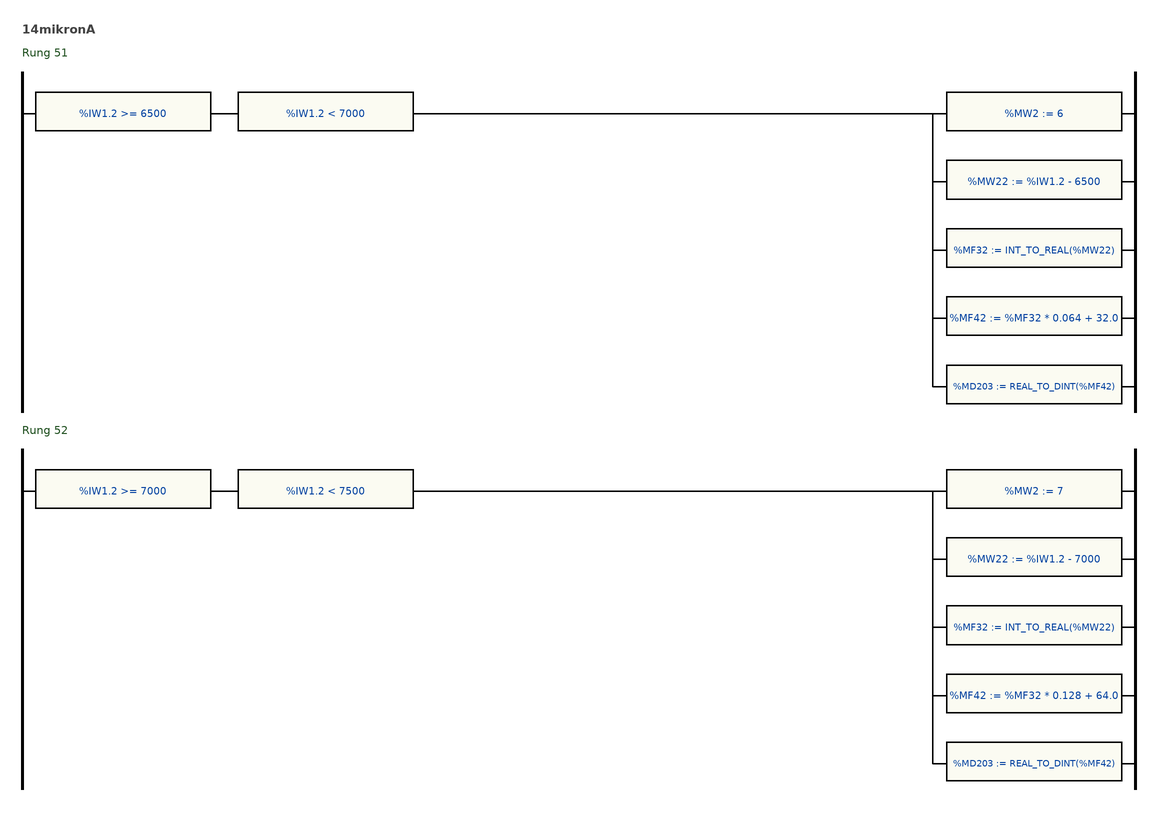
[picture p24: 14mikronA, ladder]

// Rung 51
  LD [ %IW1.2 >= 6500 ]
  AND [ %IW1.2 < 7000 ]
  [ %MW2 := 6 ]
  [ %MW22 := %IW1.2 - 6500 ]
  [ %MF32 := INT_TO_REAL ( %MW22 ) ]
  [ %MF42 := %MF32 * 0.064 + 32.0 ]
  [ %MD203 := REAL_TO_DINT ( %MF42 ) ]
  // as ST:
  //   IF %IW1.2 >= 6500 AND %IW1.2 < 7000 THEN %MW2 := 6; END_IF;
  //   IF %IW1.2 >= 6500 AND %IW1.2 < 7000 THEN %MW22 := %IW1.2 - 6500; END_IF;
  //   IF %IW1.2 >= 6500 AND %IW1.2 < 7000 THEN %MF32 := INT_TO_REAL ( %MW22 ); END_IF;
  //   IF %IW1.2 >= 6500 AND %IW1.2 < 7000 THEN %MF42 := %MF32 * 0.064 + 32.0; END_IF;
  //   IF %IW1.2 >= 6500 AND %IW1.2 < 7000 THEN %MD203 := REAL_TO_DINT ( %MF42 ); END_IF;

// Rung 52
  LD [ %IW1.2 >= 7000 ]
  AND [ %IW1.2 < 7500 ]
  [ %MW2 := 7 ]
  [ %MW22 := %IW1.2 - 7000 ]
  [ %MF32 := INT_TO_REAL ( %MW22 ) ]
  [ %MF42 := %MF32 * 0.128 + 64.0 ]
  [ %MD203 := REAL_TO_DINT ( %MF42 ) ]
  // as ST:
  //   IF %IW1.2 >= 7000 AND %IW1.2 < 7500 THEN %MW2 := 7; END_IF;
  //   IF %IW1.2 >= 7000 AND %IW1.2 < 7500 THEN %MW22 := %IW1.2 - 7000; END_IF;
  //   IF %IW1.2 >= 7000 AND %IW1.2 < 7500 THEN %MF32 := INT_TO_REAL ( %MW22 ); END_IF;
  //   IF %IW1.2 >= 7000 AND %IW1.2 < 7500 THEN %MF42 := %MF32 * 0.128 + 64.0; END_IF;
  //   IF %IW1.2 >= 7000 AND %IW1.2 < 7500 THEN %MD203 := REAL_TO_DINT ( %MF42 ); END_IF;

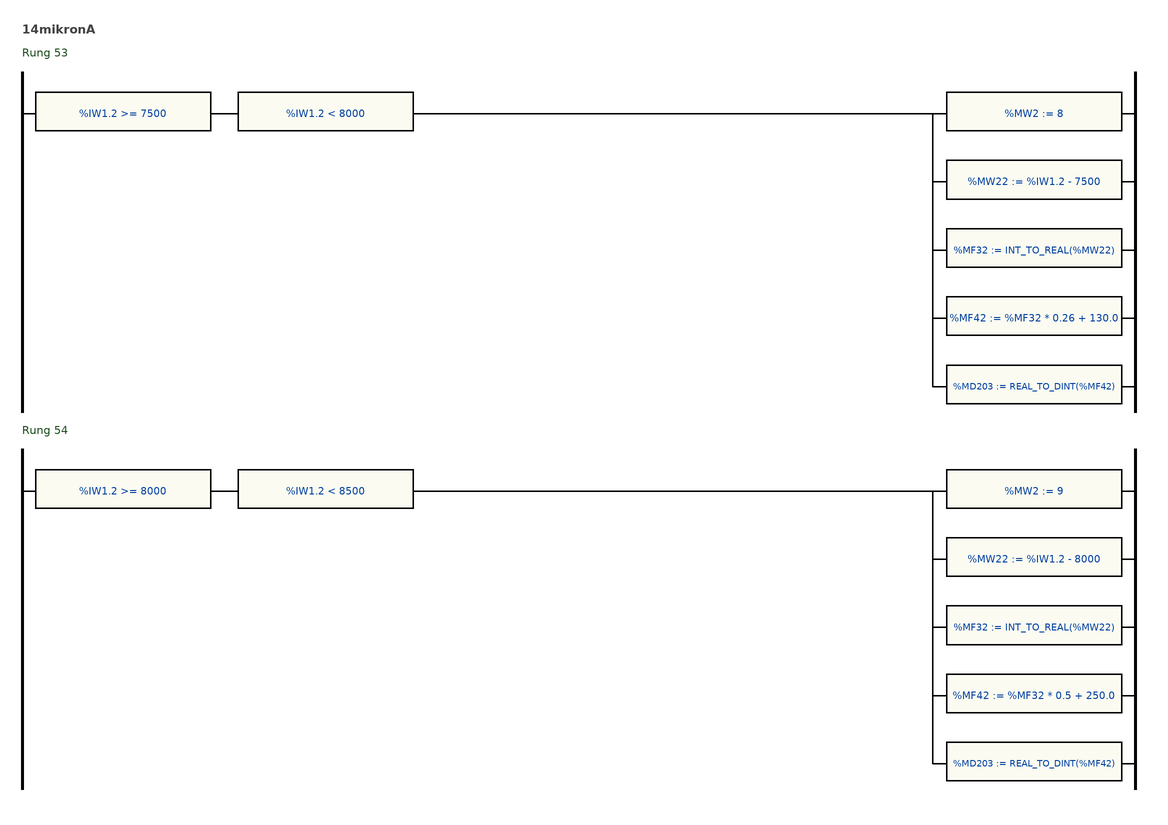

// Rung 53
  LD [ %IW1.2 >= 7500 ]
  AND [ %IW1.2 < 8000 ]
  [ %MW2 := 8 ]
  [ %MW22 := %IW1.2 - 7500 ]
  [ %MF32 := INT_TO_REAL ( %MW22 ) ]
  [ %MF42 := %MF32 * 0.26 + 130.0 ]
  [ %MD203 := REAL_TO_DINT ( %MF42 ) ]
  // as ST:
  //   IF %IW1.2 >= 7500 AND %IW1.2 < 8000 THEN %MW2 := 8; END_IF;
  //   IF %IW1.2 >= 7500 AND %IW1.2 < 8000 THEN %MW22 := %IW1.2 - 7500; END_IF;
  //   IF %IW1.2 >= 7500 AND %IW1.2 < 8000 THEN %MF32 := INT_TO_REAL ( %MW22 ); END_IF;
  //   IF %IW1.2 >= 7500 AND %IW1.2 < 8000 THEN %MF42 := %MF32 * 0.26 + 130.0; END_IF;
  //   IF %IW1.2 >= 7500 AND %IW1.2 < 8000 THEN %MD203 := REAL_TO_DINT ( %MF42 ); END_IF;

// Rung 54
  LD [ %IW1.2 >= 8000 ]
  AND [ %IW1.2 < 8500 ]
  [ %MW2 := 9 ]
  [ %MW22 := %IW1.2 - 8000 ]
  [ %MF32 := INT_TO_REAL ( %MW22 ) ]
  [ %MF42 := %MF32 * 0.5 + 250.0 ]
  [ %MD203 := REAL_TO_DINT ( %MF42 ) ]
  // as ST:
  //   IF %IW1.2 >= 8000 AND %IW1.2 < 8500 THEN %MW2 := 9; END_IF;
  //   IF %IW1.2 >= 8000 AND %IW1.2 < 8500 THEN %MW22 := %IW1.2 - 8000; END_IF;
  //   IF %IW1.2 >= 8000 AND %IW1.2 < 8500 THEN %MF32 := INT_TO_REAL ( %MW22 ); END_IF;
  //   IF %IW1.2 >= 8000 AND %IW1.2 < 8500 THEN %MF42 := %MF32 * 0.5 + 250.0; END_IF;
  //   IF %IW1.2 >= 8000 AND %IW1.2 < 8500 THEN %MD203 := REAL_TO_DINT ( %MF42 ); END_IF;

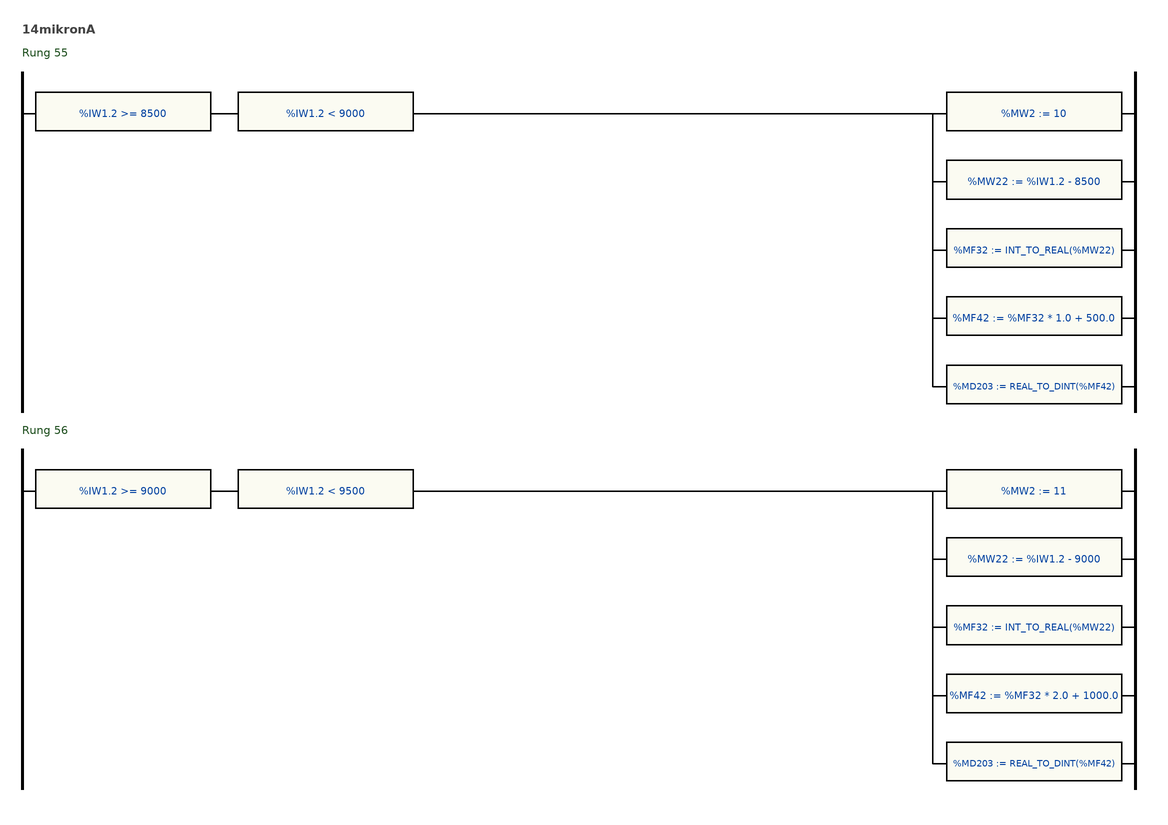

// Rung 55
  LD [ %IW1.2 >= 8500 ]
  AND [ %IW1.2 < 9000 ]
  [ %MW2 := 10 ]
  [ %MW22 := %IW1.2 - 8500 ]
  [ %MF32 := INT_TO_REAL ( %MW22 ) ]
  [ %MF42 := %MF32 * 1.0 + 500.0 ]
  [ %MD203 := REAL_TO_DINT ( %MF42 ) ]
  // as ST:
  //   IF %IW1.2 >= 8500 AND %IW1.2 < 9000 THEN %MW2 := 10; END_IF;
  //   IF %IW1.2 >= 8500 AND %IW1.2 < 9000 THEN %MW22 := %IW1.2 - 8500; END_IF;
  //   IF %IW1.2 >= 8500 AND %IW1.2 < 9000 THEN %MF32 := INT_TO_REAL ( %MW22 ); END_IF;
  //   IF %IW1.2 >= 8500 AND %IW1.2 < 9000 THEN %MF42 := %MF32 * 1.0 + 500.0; END_IF;
  //   IF %IW1.2 >= 8500 AND %IW1.2 < 9000 THEN %MD203 := REAL_TO_DINT ( %MF42 ); END_IF;

// Rung 56
  LD [ %IW1.2 >= 9000 ]
  AND [ %IW1.2 < 9500 ]
  [ %MW2 := 11 ]
  [ %MW22 := %IW1.2 - 9000 ]
  [ %MF32 := INT_TO_REAL ( %MW22 ) ]
  [ %MF42 := %MF32 * 2.0 + 1000.0 ]
  [ %MD203 := REAL_TO_DINT ( %MF42 ) ]
  // as ST:
  //   IF %IW1.2 >= 9000 AND %IW1.2 < 9500 THEN %MW2 := 11; END_IF;
  //   IF %IW1.2 >= 9000 AND %IW1.2 < 9500 THEN %MW22 := %IW1.2 - 9000; END_IF;
  //   IF %IW1.2 >= 9000 AND %IW1.2 < 9500 THEN %MF32 := INT_TO_REAL ( %MW22 ); END_IF;
  //   IF %IW1.2 >= 9000 AND %IW1.2 < 9500 THEN %MF42 := %MF32 * 2.0 + 1000.0; END_IF;
  //   IF %IW1.2 >= 9000 AND %IW1.2 < 9500 THEN %MD203 := REAL_TO_DINT ( %MF42 ); END_IF;

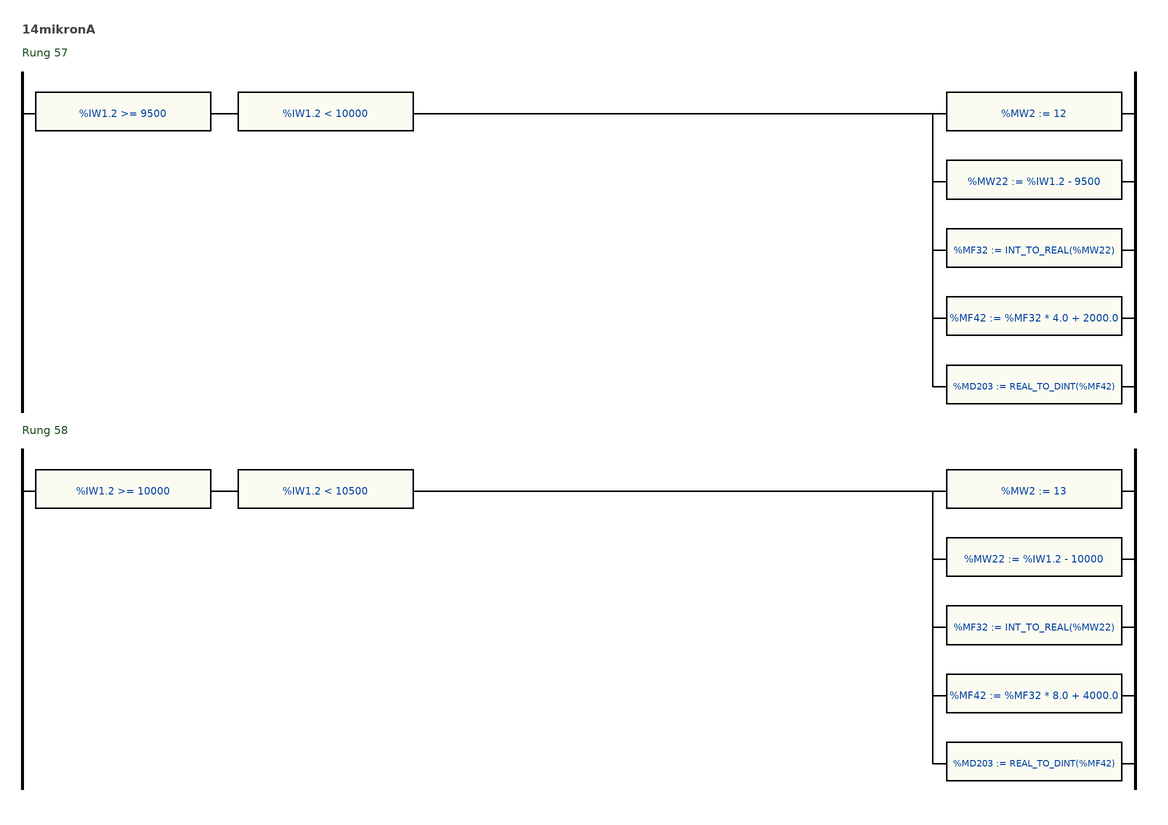

// Rung 57
  LD [ %IW1.2 >= 9500 ]
  AND [ %IW1.2 < 10000 ]
  [ %MW2 := 12 ]
  [ %MW22 := %IW1.2 - 9500 ]
  [ %MF32 := INT_TO_REAL ( %MW22 ) ]
  [ %MF42 := %MF32 * 4.0 + 2000.0 ]
  [ %MD203 := REAL_TO_DINT ( %MF42 ) ]
  // as ST:
  //   IF %IW1.2 >= 9500 AND %IW1.2 < 10000 THEN %MW2 := 12; END_IF;
  //   IF %IW1.2 >= 9500 AND %IW1.2 < 10000 THEN %MW22 := %IW1.2 - 9500; END_IF;
  //   IF %IW1.2 >= 9500 AND %IW1.2 < 10000 THEN %MF32 := INT_TO_REAL ( %MW22 ); END_IF;
  //   IF %IW1.2 >= 9500 AND %IW1.2 < 10000 THEN %MF42 := %MF32 * 4.0 + 2000.0; END_IF;
  //   IF %IW1.2 >= 9500 AND %IW1.2 < 10000 THEN %MD203 := REAL_TO_DINT ( %MF42 ); END_IF;

// Rung 58
  LD [ %IW1.2 >= 10000 ]
  AND [ %IW1.2 < 10500 ]
  [ %MW2 := 13 ]
  [ %MW22 := %IW1.2 - 10000 ]
  [ %MF32 := INT_TO_REAL ( %MW22 ) ]
  [ %MF42 := %MF32 * 8.0 + 4000.0 ]
  [ %MD203 := REAL_TO_DINT ( %MF42 ) ]
  // as ST:
  //   IF %IW1.2 >= 10000 AND %IW1.2 < 10500 THEN %MW2 := 13; END_IF;
  //   IF %IW1.2 >= 10000 AND %IW1.2 < 10500 THEN %MW22 := %IW1.2 - 10000; END_IF;
  //   IF %IW1.2 >= 10000 AND %IW1.2 < 10500 THEN %MF32 := INT_TO_REAL ( %MW22 ); END_IF;
  //   IF %IW1.2 >= 10000 AND %IW1.2 < 10500 THEN %MF42 := %MF32 * 8.0 + 4000.0; END_IF;
  //   IF %IW1.2 >= 10000 AND %IW1.2 < 10500 THEN %MD203 := REAL_TO_DINT ( %MF42 ); END_IF;

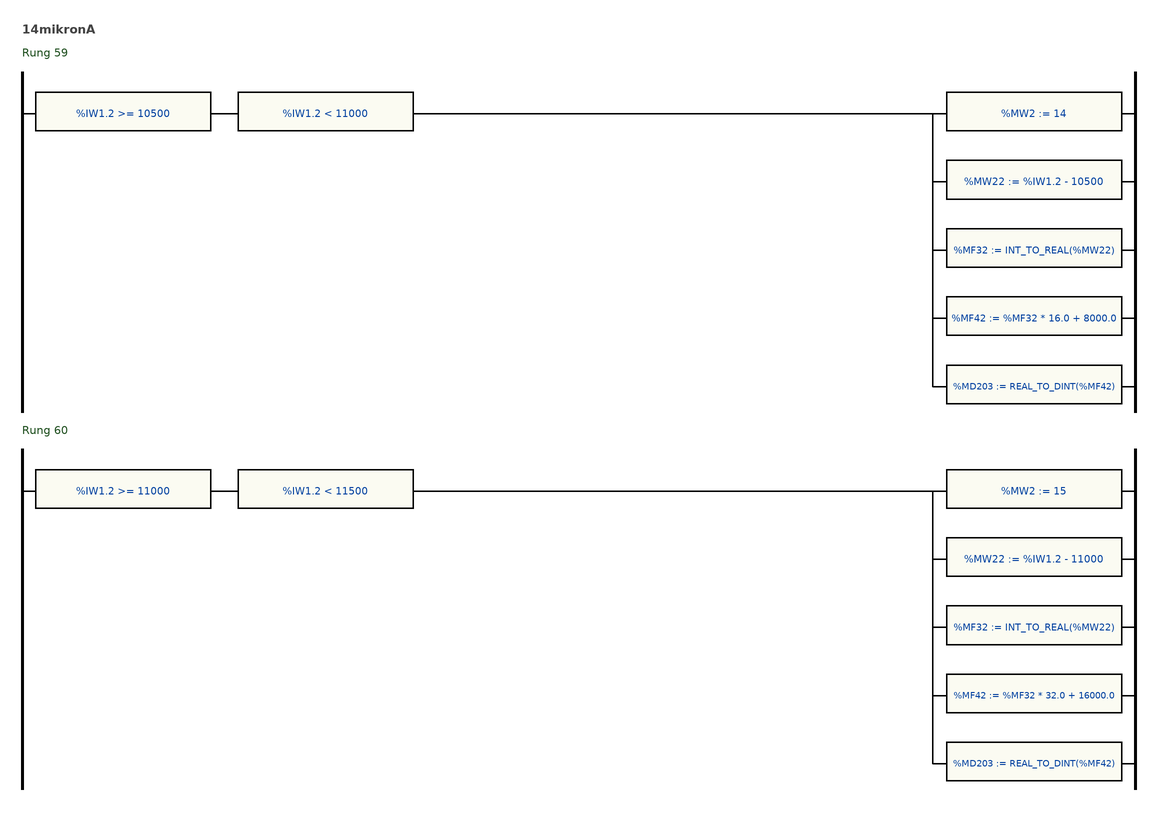

// Rung 59
  LD [ %IW1.2 >= 10500 ]
  AND [ %IW1.2 < 11000 ]
  [ %MW2 := 14 ]
  [ %MW22 := %IW1.2 - 10500 ]
  [ %MF32 := INT_TO_REAL ( %MW22 ) ]
  [ %MF42 := %MF32 * 16.0 + 8000.0 ]
  [ %MD203 := REAL_TO_DINT ( %MF42 ) ]
  // as ST:
  //   IF %IW1.2 >= 10500 AND %IW1.2 < 11000 THEN %MW2 := 14; END_IF;
  //   IF %IW1.2 >= 10500 AND %IW1.2 < 11000 THEN %MW22 := %IW1.2 - 10500; END_IF;
  //   IF %IW1.2 >= 10500 AND %IW1.2 < 11000 THEN %MF32 := INT_TO_REAL ( %MW22 ); END_IF;
  //   IF %IW1.2 >= 10500 AND %IW1.2 < 11000 THEN %MF42 := %MF32 * 16.0 + 8000.0; END_IF;
  //   IF %IW1.2 >= 10500 AND %IW1.2 < 11000 THEN %MD203 := REAL_TO_DINT ( %MF42 ); END_IF;

// Rung 60
  LD [ %IW1.2 >= 11000 ]
  AND [ %IW1.2 < 11500 ]
  [ %MW2 := 15 ]
  [ %MW22 := %IW1.2 - 11000 ]
  [ %MF32 := INT_TO_REAL ( %MW22 ) ]
  [ %MF42 := %MF32 * 32.0 + 16000.0 ]
  [ %MD203 := REAL_TO_DINT ( %MF42 ) ]
  // as ST:
  //   IF %IW1.2 >= 11000 AND %IW1.2 < 11500 THEN %MW2 := 15; END_IF;
  //   IF %IW1.2 >= 11000 AND %IW1.2 < 11500 THEN %MW22 := %IW1.2 - 11000; END_IF;
  //   IF %IW1.2 >= 11000 AND %IW1.2 < 11500 THEN %MF32 := INT_TO_REAL ( %MW22 ); END_IF;
  //   IF %IW1.2 >= 11000 AND %IW1.2 < 11500 THEN %MF42 := %MF32 * 32.0 + 16000.0; END_IF;
  //   IF %IW1.2 >= 11000 AND %IW1.2 < 11500 THEN %MD203 := REAL_TO_DINT ( %MF42 ); END_IF;

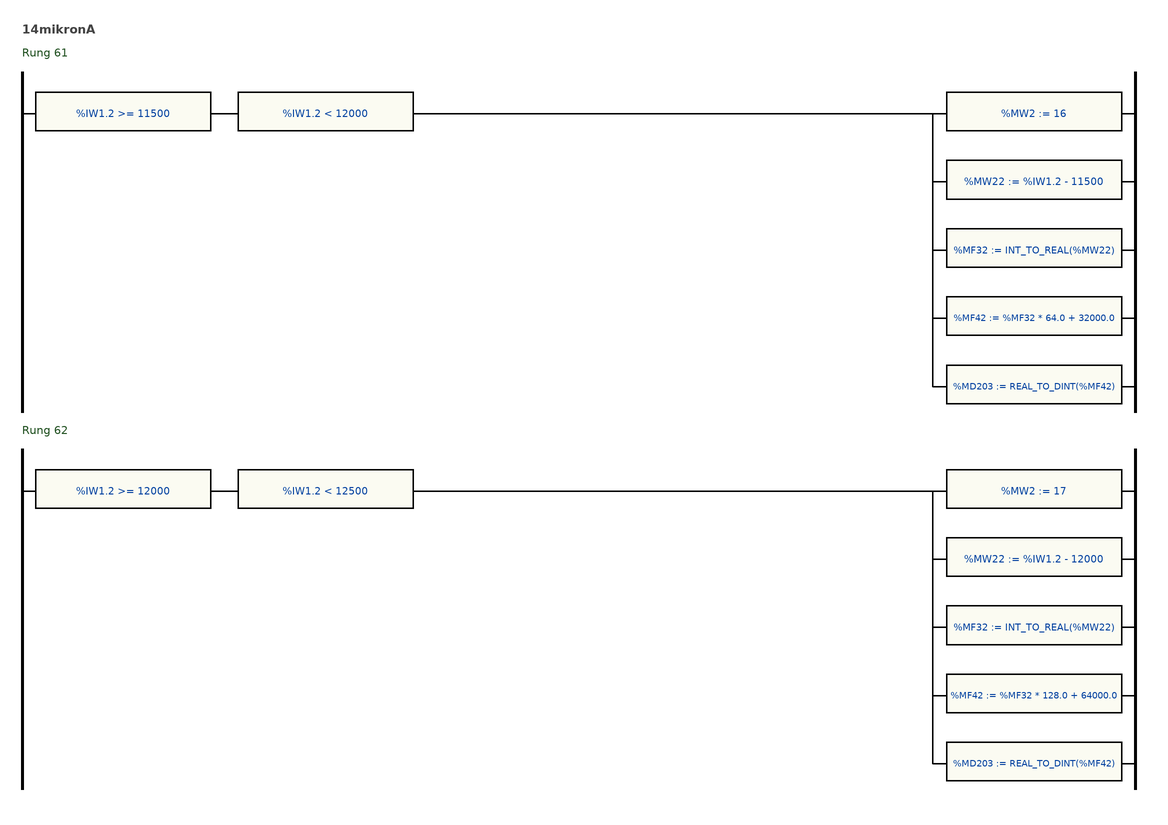

// Rung 61
  LD [ %IW1.2 >= 11500 ]
  AND [ %IW1.2 < 12000 ]
  [ %MW2 := 16 ]
  [ %MW22 := %IW1.2 - 11500 ]
  [ %MF32 := INT_TO_REAL ( %MW22 ) ]
  [ %MF42 := %MF32 * 64.0 + 32000.0 ]
  [ %MD203 := REAL_TO_DINT ( %MF42 ) ]
  // as ST:
  //   IF %IW1.2 >= 11500 AND %IW1.2 < 12000 THEN %MW2 := 16; END_IF;
  //   IF %IW1.2 >= 11500 AND %IW1.2 < 12000 THEN %MW22 := %IW1.2 - 11500; END_IF;
  //   IF %IW1.2 >= 11500 AND %IW1.2 < 12000 THEN %MF32 := INT_TO_REAL ( %MW22 ); END_IF;
  //   IF %IW1.2 >= 11500 AND %IW1.2 < 12000 THEN %MF42 := %MF32 * 64.0 + 32000.0; END_IF;
  //   IF %IW1.2 >= 11500 AND %IW1.2 < 12000 THEN %MD203 := REAL_TO_DINT ( %MF42 ); END_IF;

// Rung 62
  LD [ %IW1.2 >= 12000 ]
  AND [ %IW1.2 < 12500 ]
  [ %MW2 := 17 ]
  [ %MW22 := %IW1.2 - 12000 ]
  [ %MF32 := INT_TO_REAL ( %MW22 ) ]
  [ %MF42 := %MF32 * 128.0 + 64000.0 ]
  [ %MD203 := REAL_TO_DINT ( %MF42 ) ]
  // as ST:
  //   IF %IW1.2 >= 12000 AND %IW1.2 < 12500 THEN %MW2 := 17; END_IF;
  //   IF %IW1.2 >= 12000 AND %IW1.2 < 12500 THEN %MW22 := %IW1.2 - 12000; END_IF;
  //   IF %IW1.2 >= 12000 AND %IW1.2 < 12500 THEN %MF32 := INT_TO_REAL ( %MW22 ); END_IF;
  //   IF %IW1.2 >= 12000 AND %IW1.2 < 12500 THEN %MF42 := %MF32 * 128.0 + 64000.0; END_IF;
  //   IF %IW1.2 >= 12000 AND %IW1.2 < 12500 THEN %MD203 := REAL_TO_DINT ( %MF42 ); END_IF;

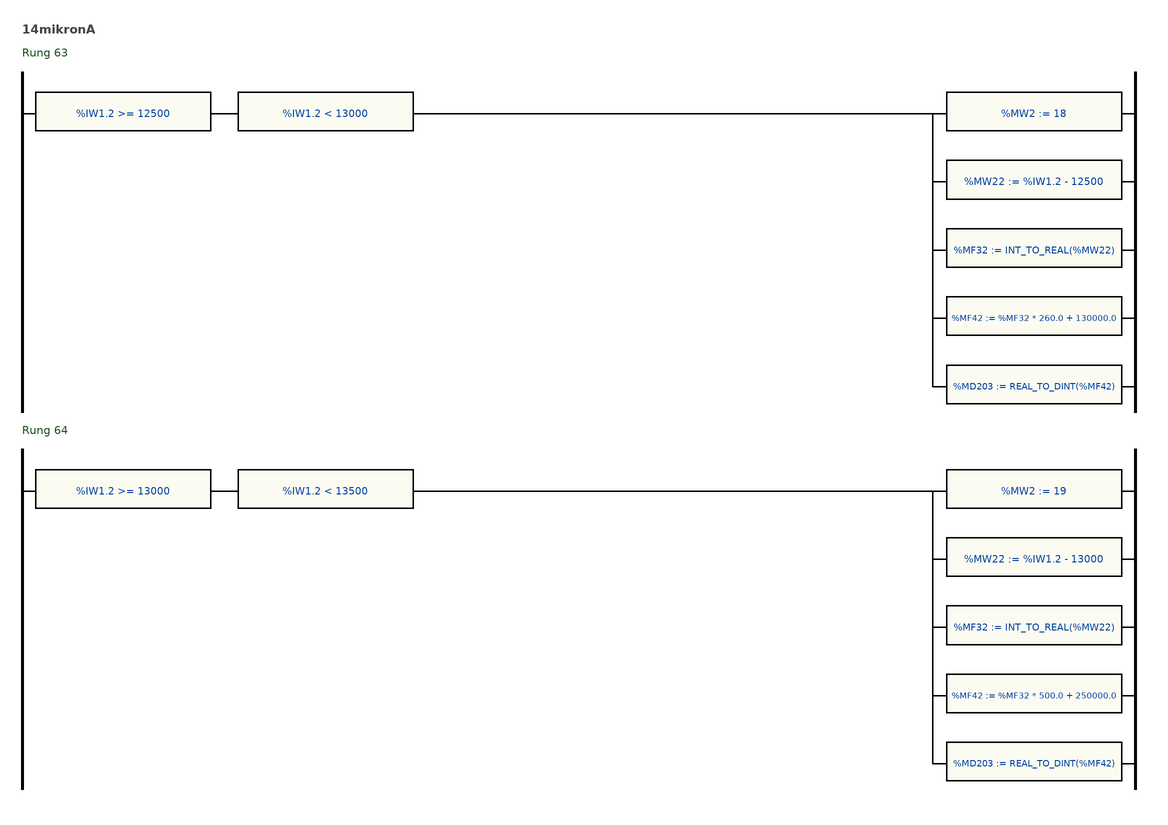

// Rung 63
  LD [ %IW1.2 >= 12500 ]
  AND [ %IW1.2 < 13000 ]
  [ %MW2 := 18 ]
  [ %MW22 := %IW1.2 - 12500 ]
  [ %MF32 := INT_TO_REAL ( %MW22 ) ]
  [ %MF42 := %MF32 * 260.0 + 130000.0 ]
  [ %MD203 := REAL_TO_DINT ( %MF42 ) ]
  // as ST:
  //   IF %IW1.2 >= 12500 AND %IW1.2 < 13000 THEN %MW2 := 18; END_IF;
  //   IF %IW1.2 >= 12500 AND %IW1.2 < 13000 THEN %MW22 := %IW1.2 - 12500; END_IF;
  //   IF %IW1.2 >= 12500 AND %IW1.2 < 13000 THEN %MF32 := INT_TO_REAL ( %MW22 ); END_IF;
  //   IF %IW1.2 >= 12500 AND %IW1.2 < 13000 THEN %MF42 := %MF32 * 260.0 + 130000.0; END_IF;
  //   IF %IW1.2 >= 12500 AND %IW1.2 < 13000 THEN %MD203 := REAL_TO_DINT ( %MF42 ); END_IF;

// Rung 64
  LD [ %IW1.2 >= 13000 ]
  AND [ %IW1.2 < 13500 ]
  [ %MW2 := 19 ]
  [ %MW22 := %IW1.2 - 13000 ]
  [ %MF32 := INT_TO_REAL ( %MW22 ) ]
  [ %MF42 := %MF32 * 500.0 + 250000.0 ]
  [ %MD203 := REAL_TO_DINT ( %MF42 ) ]
  // as ST:
  //   IF %IW1.2 >= 13000 AND %IW1.2 < 13500 THEN %MW2 := 19; END_IF;
  //   IF %IW1.2 >= 13000 AND %IW1.2 < 13500 THEN %MW22 := %IW1.2 - 13000; END_IF;
  //   IF %IW1.2 >= 13000 AND %IW1.2 < 13500 THEN %MF32 := INT_TO_REAL ( %MW22 ); END_IF;
  //   IF %IW1.2 >= 13000 AND %IW1.2 < 13500 THEN %MF42 := %MF32 * 500.0 + 250000.0; END_IF;
  //   IF %IW1.2 >= 13000 AND %IW1.2 < 13500 THEN %MD203 := REAL_TO_DINT ( %MF42 ); END_IF;

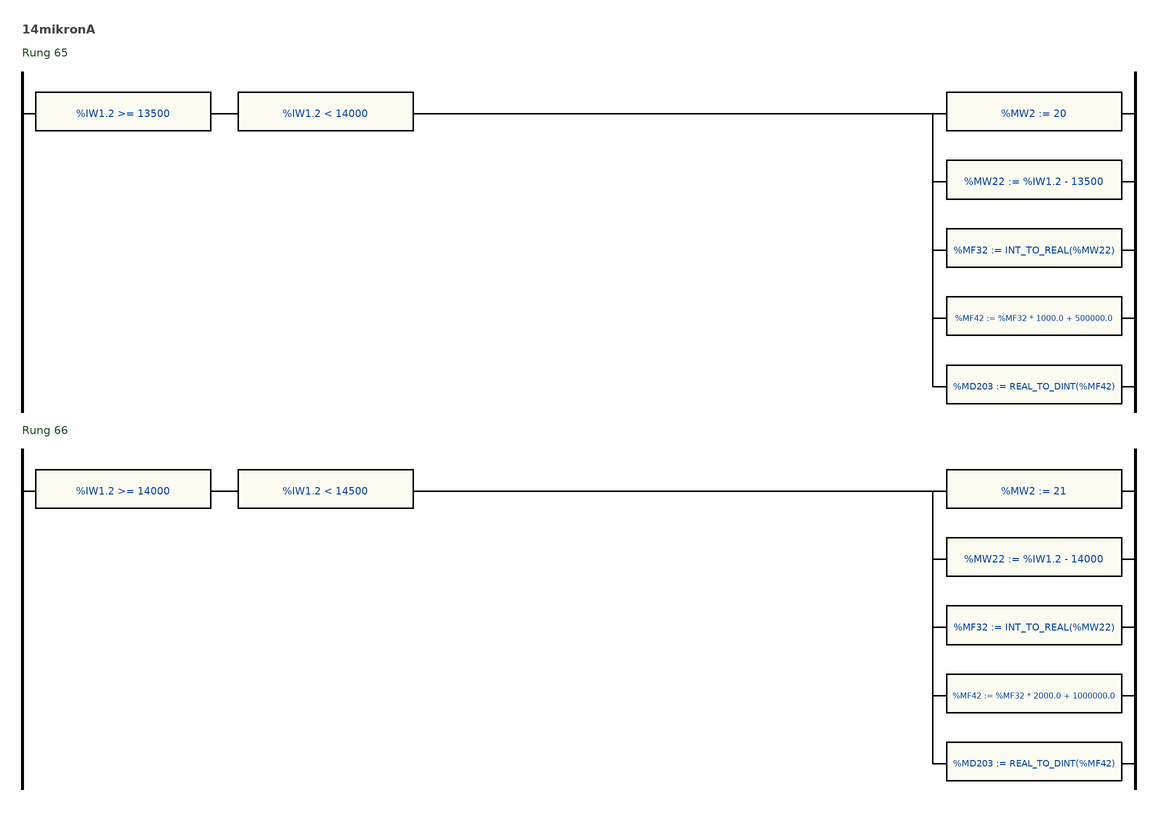

// Rung 65
  LD [ %IW1.2 >= 13500 ]
  AND [ %IW1.2 < 14000 ]
  [ %MW2 := 20 ]
  [ %MW22 := %IW1.2 - 13500 ]
  [ %MF32 := INT_TO_REAL ( %MW22 ) ]
  [ %MF42 := %MF32 * 1000.0 + 500000.0 ]
  [ %MD203 := REAL_TO_DINT ( %MF42 ) ]
  // as ST:
  //   IF %IW1.2 >= 13500 AND %IW1.2 < 14000 THEN %MW2 := 20; END_IF;
  //   IF %IW1.2 >= 13500 AND %IW1.2 < 14000 THEN %MW22 := %IW1.2 - 13500; END_IF;
  //   IF %IW1.2 >= 13500 AND %IW1.2 < 14000 THEN %MF32 := INT_TO_REAL ( %MW22 ); END_IF;
  //   IF %IW1.2 >= 13500 AND %IW1.2 < 14000 THEN %MF42 := %MF32 * 1000.0 + 500000.0; END_IF;
  //   IF %IW1.2 >= 13500 AND %IW1.2 < 14000 THEN %MD203 := REAL_TO_DINT ( %MF42 ); END_IF;

// Rung 66
  LD [ %IW1.2 >= 14000 ]
  AND [ %IW1.2 < 14500 ]
  [ %MW2 := 21 ]
  [ %MW22 := %IW1.2 - 14000 ]
  [ %MF32 := INT_TO_REAL ( %MW22 ) ]
  [ %MF42 := %MF32 * 2000.0 + 1000000.0 ]
  [ %MD203 := REAL_TO_DINT ( %MF42 ) ]
  // as ST:
  //   IF %IW1.2 >= 14000 AND %IW1.2 < 14500 THEN %MW2 := 21; END_IF;
  //   IF %IW1.2 >= 14000 AND %IW1.2 < 14500 THEN %MW22 := %IW1.2 - 14000; END_IF;
  //   IF %IW1.2 >= 14000 AND %IW1.2 < 14500 THEN %MF32 := INT_TO_REAL ( %MW22 ); END_IF;
  //   IF %IW1.2 >= 14000 AND %IW1.2 < 14500 THEN %MF42 := %MF32 * 2000.0 + 1000000.0; END_IF;
  //   IF %IW1.2 >= 14000 AND %IW1.2 < 14500 THEN %MD203 := REAL_TO_DINT ( %MF42 ); END_IF;

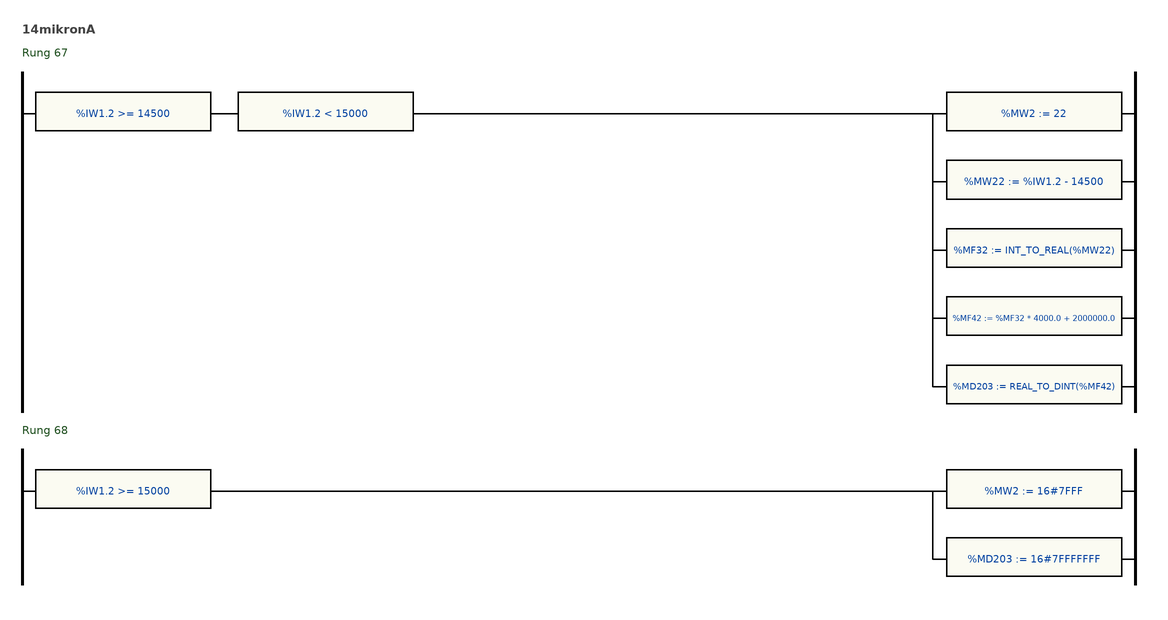

// Rung 67
  LD [ %IW1.2 >= 14500 ]
  AND [ %IW1.2 < 15000 ]
  [ %MW2 := 22 ]
  [ %MW22 := %IW1.2 - 14500 ]
  [ %MF32 := INT_TO_REAL ( %MW22 ) ]
  [ %MF42 := %MF32 * 4000.0 + 2000000.0 ]
  [ %MD203 := REAL_TO_DINT ( %MF42 ) ]
  // as ST:
  //   IF %IW1.2 >= 14500 AND %IW1.2 < 15000 THEN %MW2 := 22; END_IF;
  //   IF %IW1.2 >= 14500 AND %IW1.2 < 15000 THEN %MW22 := %IW1.2 - 14500; END_IF;
  //   IF %IW1.2 >= 14500 AND %IW1.2 < 15000 THEN %MF32 := INT_TO_REAL ( %MW22 ); END_IF;
  //   IF %IW1.2 >= 14500 AND %IW1.2 < 15000 THEN %MF42 := %MF32 * 4000.0 + 2000000.0; END_IF;
  //   IF %IW1.2 >= 14500 AND %IW1.2 < 15000 THEN %MD203 := REAL_TO_DINT ( %MF42 ); END_IF;

// Rung 68
  LD [ %IW1.2 >= 15000 ]
  [ %MW2 := 16#7FFF ]
  [ %MD203 := 16#7FFFFFFF ]
  // as ST:
  //   IF %IW1.2 >= 15000 THEN %MW2 := 16#7FFF; END_IF;
  //   IF %IW1.2 >= 15000 THEN %MD203 := 16#7FFFFFFF; END_IF;

POU 4mikronB
  (* SectionNumber=4 *)

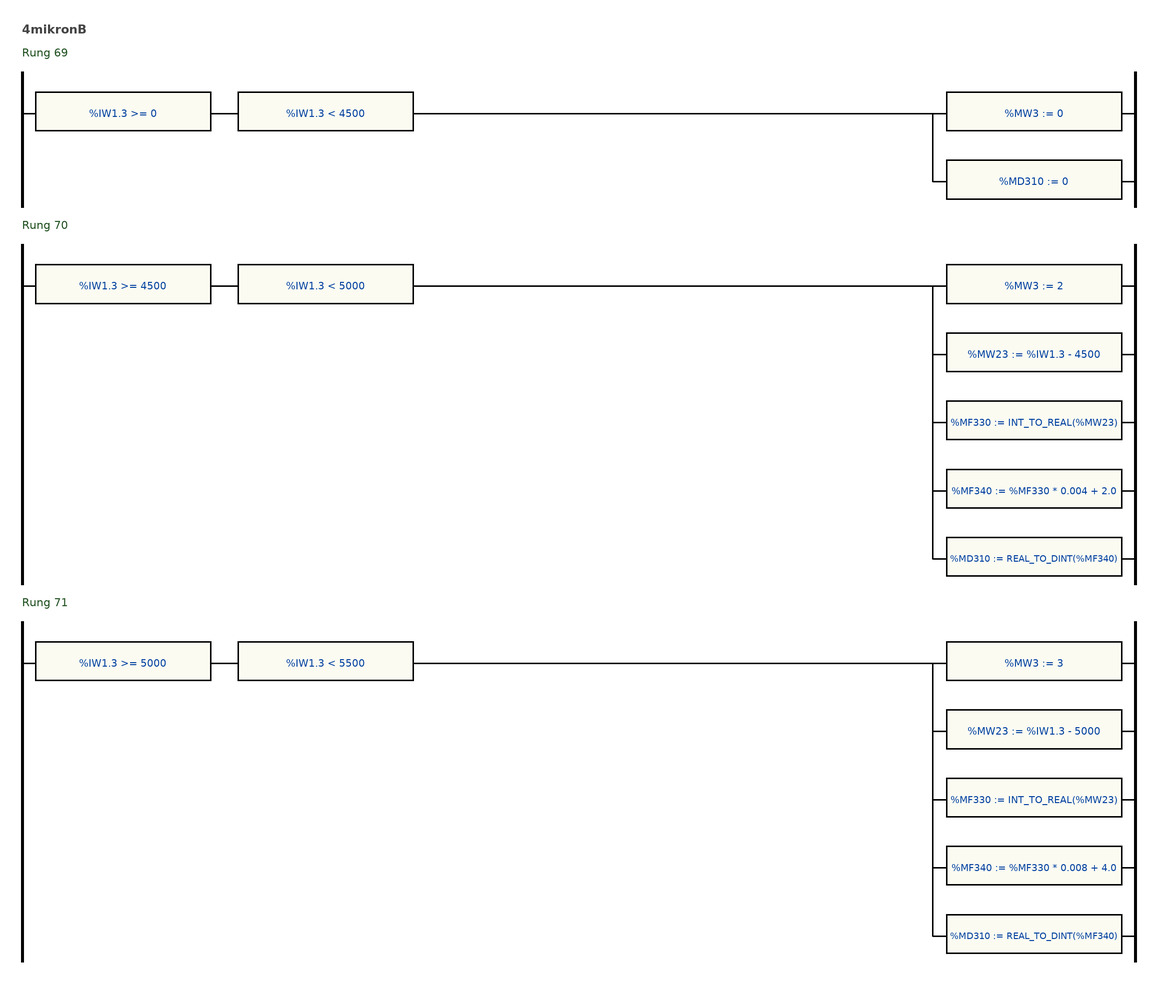

// Rung 69
  LD [ %IW1.3 >= 0 ]
  AND [ %IW1.3 < 4500 ]
  [ %MW3 := 0 ]
  [ %MD310 := 0 ]
  // as ST:
  //   IF %IW1.3 >= 0 AND %IW1.3 < 4500 THEN %MW3 := 0; END_IF;
  //   IF %IW1.3 >= 0 AND %IW1.3 < 4500 THEN %MD310 := 0; END_IF;

// Rung 70
  LD [ %IW1.3 >= 4500 ]
  AND [ %IW1.3 < 5000 ]
  [ %MW3 := 2 ]
  [ %MW23 := %IW1.3 - 4500 ]
  [ %MF330 := INT_TO_REAL ( %MW23 ) ]
  [ %MF340 := %MF330 * 0.004 + 2.0 ]
  [ %MD310 := REAL_TO_DINT ( %MF340 ) ]
  // as ST:
  //   IF %IW1.3 >= 4500 AND %IW1.3 < 5000 THEN %MW3 := 2; END_IF;
  //   IF %IW1.3 >= 4500 AND %IW1.3 < 5000 THEN %MW23 := %IW1.3 - 4500; END_IF;
  //   IF %IW1.3 >= 4500 AND %IW1.3 < 5000 THEN %MF330 := INT_TO_REAL ( %MW23 ); END_IF;
  //   IF %IW1.3 >= 4500 AND %IW1.3 < 5000 THEN %MF340 := %MF330 * 0.004 + 2.0; END_IF;
  //   IF %IW1.3 >= 4500 AND %IW1.3 < 5000 THEN %MD310 := REAL_TO_DINT ( %MF340 ); END_IF;

// Rung 71
  LD [ %IW1.3 >= 5000 ]
  AND [ %IW1.3 < 5500 ]
  [ %MW3 := 3 ]
  [ %MW23 := %IW1.3 - 5000 ]
  [ %MF330 := INT_TO_REAL ( %MW23 ) ]
  [ %MF340 := %MF330 * 0.008 + 4.0 ]
  [ %MD310 := REAL_TO_DINT ( %MF340 ) ]
  // as ST:
  //   IF %IW1.3 >= 5000 AND %IW1.3 < 5500 THEN %MW3 := 3; END_IF;
  //   IF %IW1.3 >= 5000 AND %IW1.3 < 5500 THEN %MW23 := %IW1.3 - 5000; END_IF;
  //   IF %IW1.3 >= 5000 AND %IW1.3 < 5500 THEN %MF330 := INT_TO_REAL ( %MW23 ); END_IF;
  //   IF %IW1.3 >= 5000 AND %IW1.3 < 5500 THEN %MF340 := %MF330 * 0.008 + 4.0; END_IF;
  //   IF %IW1.3 >= 5000 AND %IW1.3 < 5500 THEN %MD310 := REAL_TO_DINT ( %MF340 ); END_IF;

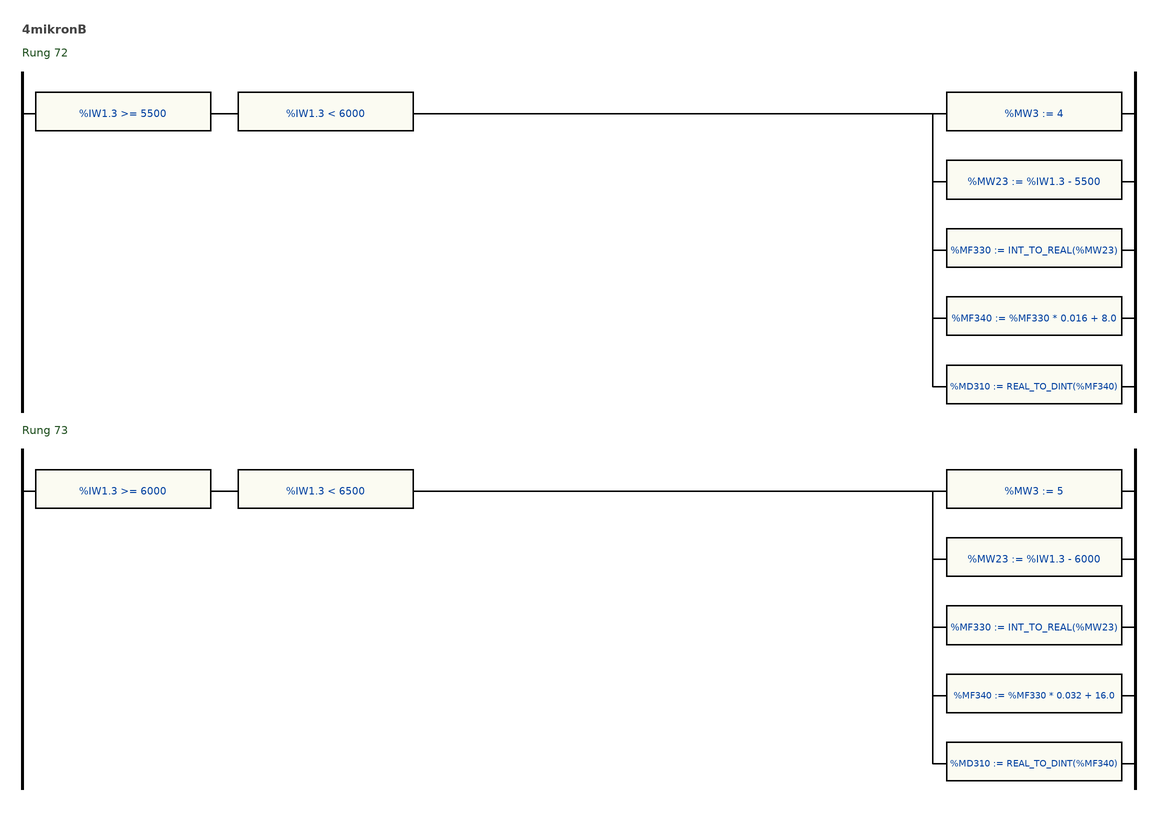

// Rung 72
  LD [ %IW1.3 >= 5500 ]
  AND [ %IW1.3 < 6000 ]
  [ %MW3 := 4 ]
  [ %MW23 := %IW1.3 - 5500 ]
  [ %MF330 := INT_TO_REAL ( %MW23 ) ]
  [ %MF340 := %MF330 * 0.016 + 8.0 ]
  [ %MD310 := REAL_TO_DINT ( %MF340 ) ]
  // as ST:
  //   IF %IW1.3 >= 5500 AND %IW1.3 < 6000 THEN %MW3 := 4; END_IF;
  //   IF %IW1.3 >= 5500 AND %IW1.3 < 6000 THEN %MW23 := %IW1.3 - 5500; END_IF;
  //   IF %IW1.3 >= 5500 AND %IW1.3 < 6000 THEN %MF330 := INT_TO_REAL ( %MW23 ); END_IF;
  //   IF %IW1.3 >= 5500 AND %IW1.3 < 6000 THEN %MF340 := %MF330 * 0.016 + 8.0; END_IF;
  //   IF %IW1.3 >= 5500 AND %IW1.3 < 6000 THEN %MD310 := REAL_TO_DINT ( %MF340 ); END_IF;

// Rung 73
  LD [ %IW1.3 >= 6000 ]
  AND [ %IW1.3 < 6500 ]
  [ %MW3 := 5 ]
  [ %MW23 := %IW1.3 - 6000 ]
  [ %MF330 := INT_TO_REAL ( %MW23 ) ]
  [ %MF340 := %MF330 * 0.032 + 16.0 ]
  [ %MD310 := REAL_TO_DINT ( %MF340 ) ]
  // as ST:
  //   IF %IW1.3 >= 6000 AND %IW1.3 < 6500 THEN %MW3 := 5; END_IF;
  //   IF %IW1.3 >= 6000 AND %IW1.3 < 6500 THEN %MW23 := %IW1.3 - 6000; END_IF;
  //   IF %IW1.3 >= 6000 AND %IW1.3 < 6500 THEN %MF330 := INT_TO_REAL ( %MW23 ); END_IF;
  //   IF %IW1.3 >= 6000 AND %IW1.3 < 6500 THEN %MF340 := %MF330 * 0.032 + 16.0; END_IF;
  //   IF %IW1.3 >= 6000 AND %IW1.3 < 6500 THEN %MD310 := REAL_TO_DINT ( %MF340 ); END_IF;

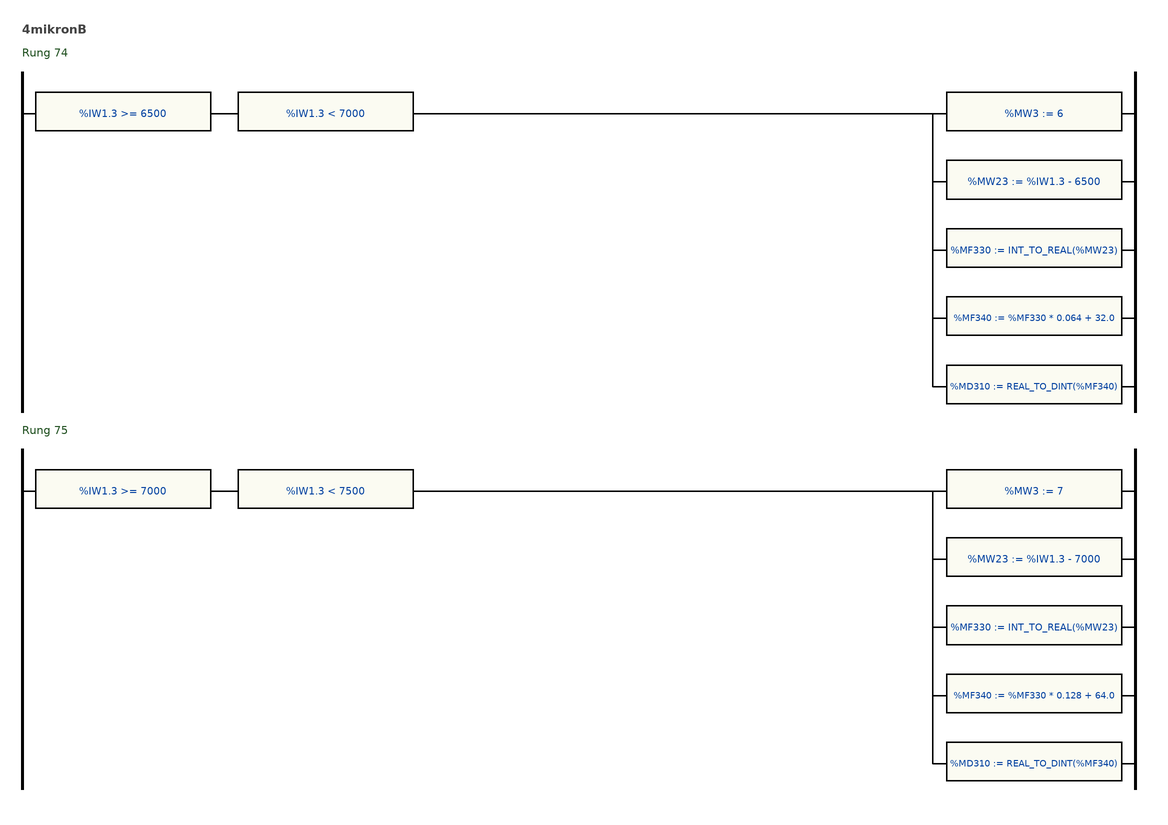

// Rung 74
  LD [ %IW1.3 >= 6500 ]
  AND [ %IW1.3 < 7000 ]
  [ %MW3 := 6 ]
  [ %MW23 := %IW1.3 - 6500 ]
  [ %MF330 := INT_TO_REAL ( %MW23 ) ]
  [ %MF340 := %MF330 * 0.064 + 32.0 ]
  [ %MD310 := REAL_TO_DINT ( %MF340 ) ]
  // as ST:
  //   IF %IW1.3 >= 6500 AND %IW1.3 < 7000 THEN %MW3 := 6; END_IF;
  //   IF %IW1.3 >= 6500 AND %IW1.3 < 7000 THEN %MW23 := %IW1.3 - 6500; END_IF;
  //   IF %IW1.3 >= 6500 AND %IW1.3 < 7000 THEN %MF330 := INT_TO_REAL ( %MW23 ); END_IF;
  //   IF %IW1.3 >= 6500 AND %IW1.3 < 7000 THEN %MF340 := %MF330 * 0.064 + 32.0; END_IF;
  //   IF %IW1.3 >= 6500 AND %IW1.3 < 7000 THEN %MD310 := REAL_TO_DINT ( %MF340 ); END_IF;

// Rung 75
  LD [ %IW1.3 >= 7000 ]
  AND [ %IW1.3 < 7500 ]
  [ %MW3 := 7 ]
  [ %MW23 := %IW1.3 - 7000 ]
  [ %MF330 := INT_TO_REAL ( %MW23 ) ]
  [ %MF340 := %MF330 * 0.128 + 64.0 ]
  [ %MD310 := REAL_TO_DINT ( %MF340 ) ]
  // as ST:
  //   IF %IW1.3 >= 7000 AND %IW1.3 < 7500 THEN %MW3 := 7; END_IF;
  //   IF %IW1.3 >= 7000 AND %IW1.3 < 7500 THEN %MW23 := %IW1.3 - 7000; END_IF;
  //   IF %IW1.3 >= 7000 AND %IW1.3 < 7500 THEN %MF330 := INT_TO_REAL ( %MW23 ); END_IF;
  //   IF %IW1.3 >= 7000 AND %IW1.3 < 7500 THEN %MF340 := %MF330 * 0.128 + 64.0; END_IF;
  //   IF %IW1.3 >= 7000 AND %IW1.3 < 7500 THEN %MD310 := REAL_TO_DINT ( %MF340 ); END_IF;

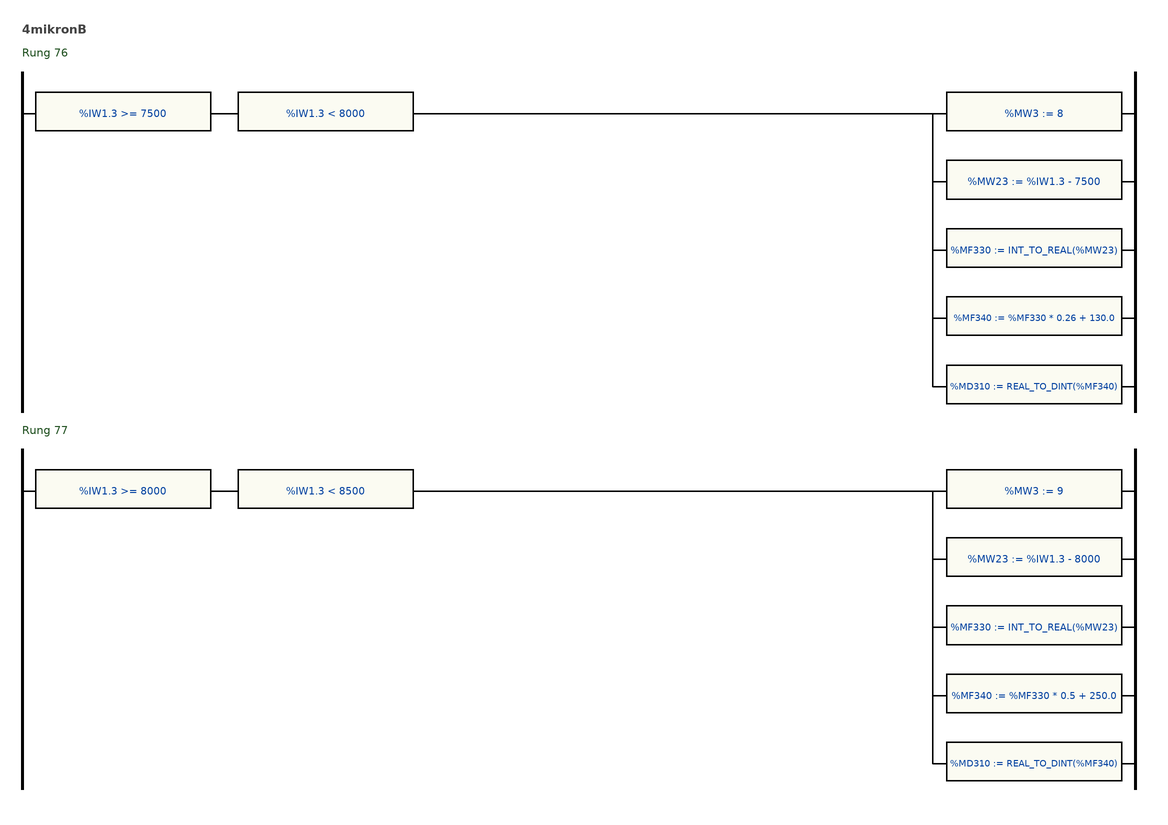

// Rung 76
  LD [ %IW1.3 >= 7500 ]
  AND [ %IW1.3 < 8000 ]
  [ %MW3 := 8 ]
  [ %MW23 := %IW1.3 - 7500 ]
  [ %MF330 := INT_TO_REAL ( %MW23 ) ]
  [ %MF340 := %MF330 * 0.26 + 130.0 ]
  [ %MD310 := REAL_TO_DINT ( %MF340 ) ]
  // as ST:
  //   IF %IW1.3 >= 7500 AND %IW1.3 < 8000 THEN %MW3 := 8; END_IF;
  //   IF %IW1.3 >= 7500 AND %IW1.3 < 8000 THEN %MW23 := %IW1.3 - 7500; END_IF;
  //   IF %IW1.3 >= 7500 AND %IW1.3 < 8000 THEN %MF330 := INT_TO_REAL ( %MW23 ); END_IF;
  //   IF %IW1.3 >= 7500 AND %IW1.3 < 8000 THEN %MF340 := %MF330 * 0.26 + 130.0; END_IF;
  //   IF %IW1.3 >= 7500 AND %IW1.3 < 8000 THEN %MD310 := REAL_TO_DINT ( %MF340 ); END_IF;

// Rung 77
  LD [ %IW1.3 >= 8000 ]
  AND [ %IW1.3 < 8500 ]
  [ %MW3 := 9 ]
  [ %MW23 := %IW1.3 - 8000 ]
  [ %MF330 := INT_TO_REAL ( %MW23 ) ]
  [ %MF340 := %MF330 * 0.5 + 250.0 ]
  [ %MD310 := REAL_TO_DINT ( %MF340 ) ]
  // as ST:
  //   IF %IW1.3 >= 8000 AND %IW1.3 < 8500 THEN %MW3 := 9; END_IF;
  //   IF %IW1.3 >= 8000 AND %IW1.3 < 8500 THEN %MW23 := %IW1.3 - 8000; END_IF;
  //   IF %IW1.3 >= 8000 AND %IW1.3 < 8500 THEN %MF330 := INT_TO_REAL ( %MW23 ); END_IF;
  //   IF %IW1.3 >= 8000 AND %IW1.3 < 8500 THEN %MF340 := %MF330 * 0.5 + 250.0; END_IF;
  //   IF %IW1.3 >= 8000 AND %IW1.3 < 8500 THEN %MD310 := REAL_TO_DINT ( %MF340 ); END_IF;

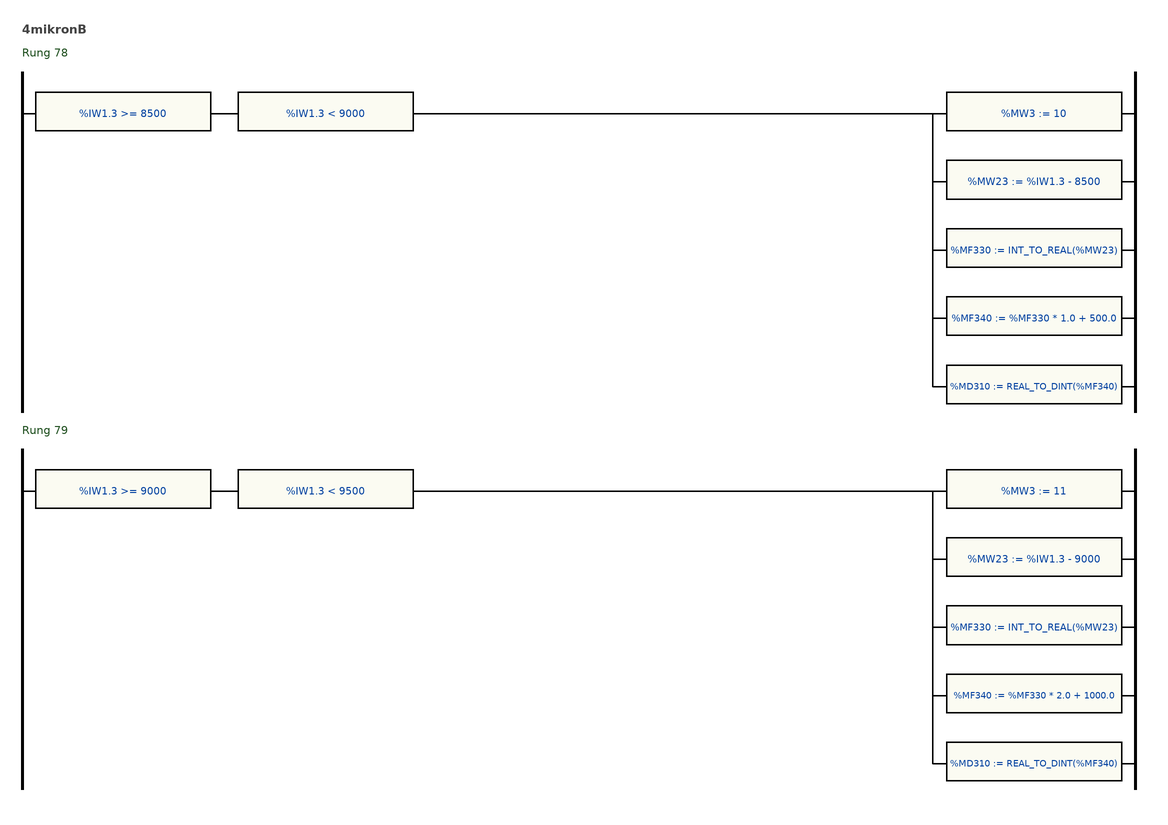

// Rung 78
  LD [ %IW1.3 >= 8500 ]
  AND [ %IW1.3 < 9000 ]
  [ %MW3 := 10 ]
  [ %MW23 := %IW1.3 - 8500 ]
  [ %MF330 := INT_TO_REAL ( %MW23 ) ]
  [ %MF340 := %MF330 * 1.0 + 500.0 ]
  [ %MD310 := REAL_TO_DINT ( %MF340 ) ]
  // as ST:
  //   IF %IW1.3 >= 8500 AND %IW1.3 < 9000 THEN %MW3 := 10; END_IF;
  //   IF %IW1.3 >= 8500 AND %IW1.3 < 9000 THEN %MW23 := %IW1.3 - 8500; END_IF;
  //   IF %IW1.3 >= 8500 AND %IW1.3 < 9000 THEN %MF330 := INT_TO_REAL ( %MW23 ); END_IF;
  //   IF %IW1.3 >= 8500 AND %IW1.3 < 9000 THEN %MF340 := %MF330 * 1.0 + 500.0; END_IF;
  //   IF %IW1.3 >= 8500 AND %IW1.3 < 9000 THEN %MD310 := REAL_TO_DINT ( %MF340 ); END_IF;

// Rung 79
  LD [ %IW1.3 >= 9000 ]
  AND [ %IW1.3 < 9500 ]
  [ %MW3 := 11 ]
  [ %MW23 := %IW1.3 - 9000 ]
  [ %MF330 := INT_TO_REAL ( %MW23 ) ]
  [ %MF340 := %MF330 * 2.0 + 1000.0 ]
  [ %MD310 := REAL_TO_DINT ( %MF340 ) ]
  // as ST:
  //   IF %IW1.3 >= 9000 AND %IW1.3 < 9500 THEN %MW3 := 11; END_IF;
  //   IF %IW1.3 >= 9000 AND %IW1.3 < 9500 THEN %MW23 := %IW1.3 - 9000; END_IF;
  //   IF %IW1.3 >= 9000 AND %IW1.3 < 9500 THEN %MF330 := INT_TO_REAL ( %MW23 ); END_IF;
  //   IF %IW1.3 >= 9000 AND %IW1.3 < 9500 THEN %MF340 := %MF330 * 2.0 + 1000.0; END_IF;
  //   IF %IW1.3 >= 9000 AND %IW1.3 < 9500 THEN %MD310 := REAL_TO_DINT ( %MF340 ); END_IF;

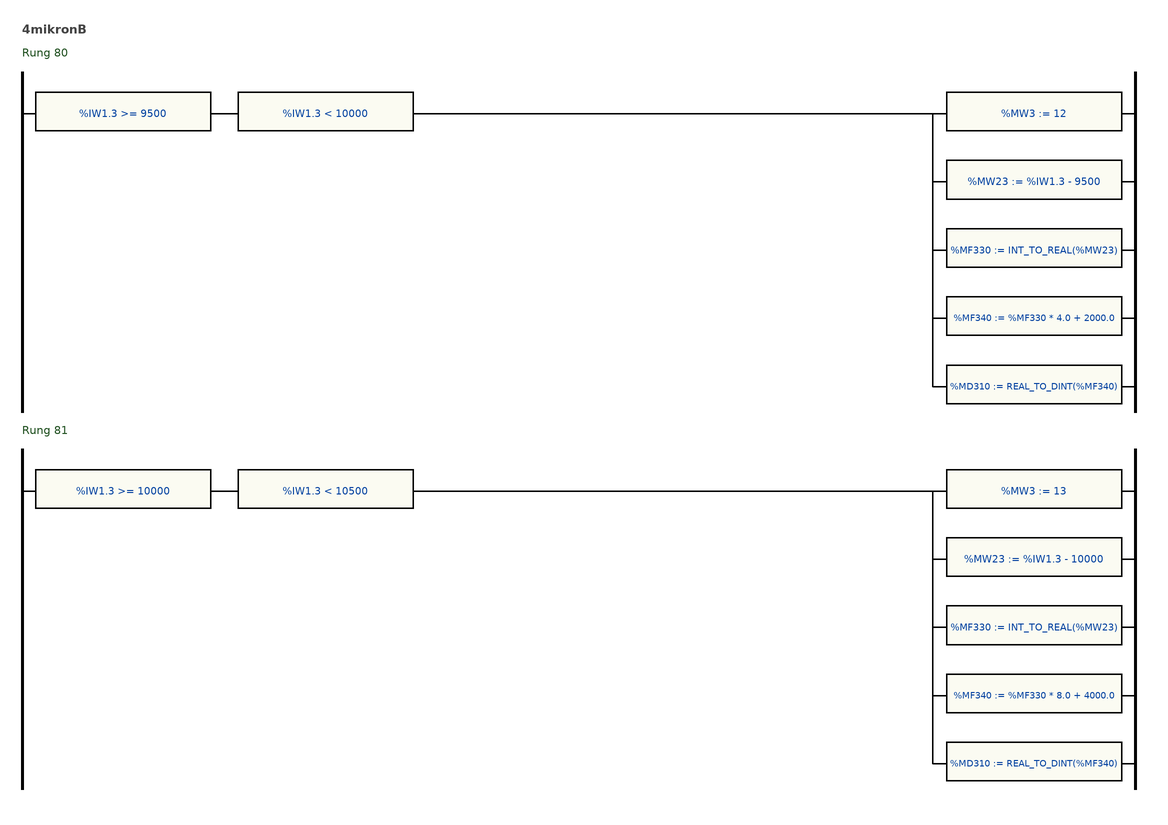

// Rung 80
  LD [ %IW1.3 >= 9500 ]
  AND [ %IW1.3 < 10000 ]
  [ %MW3 := 12 ]
  [ %MW23 := %IW1.3 - 9500 ]
  [ %MF330 := INT_TO_REAL ( %MW23 ) ]
  [ %MF340 := %MF330 * 4.0 + 2000.0 ]
  [ %MD310 := REAL_TO_DINT ( %MF340 ) ]
  // as ST:
  //   IF %IW1.3 >= 9500 AND %IW1.3 < 10000 THEN %MW3 := 12; END_IF;
  //   IF %IW1.3 >= 9500 AND %IW1.3 < 10000 THEN %MW23 := %IW1.3 - 9500; END_IF;
  //   IF %IW1.3 >= 9500 AND %IW1.3 < 10000 THEN %MF330 := INT_TO_REAL ( %MW23 ); END_IF;
  //   IF %IW1.3 >= 9500 AND %IW1.3 < 10000 THEN %MF340 := %MF330 * 4.0 + 2000.0; END_IF;
  //   IF %IW1.3 >= 9500 AND %IW1.3 < 10000 THEN %MD310 := REAL_TO_DINT ( %MF340 ); END_IF;

// Rung 81
  LD [ %IW1.3 >= 10000 ]
  AND [ %IW1.3 < 10500 ]
  [ %MW3 := 13 ]
  [ %MW23 := %IW1.3 - 10000 ]
  [ %MF330 := INT_TO_REAL ( %MW23 ) ]
  [ %MF340 := %MF330 * 8.0 + 4000.0 ]
  [ %MD310 := REAL_TO_DINT ( %MF340 ) ]
  // as ST:
  //   IF %IW1.3 >= 10000 AND %IW1.3 < 10500 THEN %MW3 := 13; END_IF;
  //   IF %IW1.3 >= 10000 AND %IW1.3 < 10500 THEN %MW23 := %IW1.3 - 10000; END_IF;
  //   IF %IW1.3 >= 10000 AND %IW1.3 < 10500 THEN %MF330 := INT_TO_REAL ( %MW23 ); END_IF;
  //   IF %IW1.3 >= 10000 AND %IW1.3 < 10500 THEN %MF340 := %MF330 * 8.0 + 4000.0; END_IF;
  //   IF %IW1.3 >= 10000 AND %IW1.3 < 10500 THEN %MD310 := REAL_TO_DINT ( %MF340 ); END_IF;

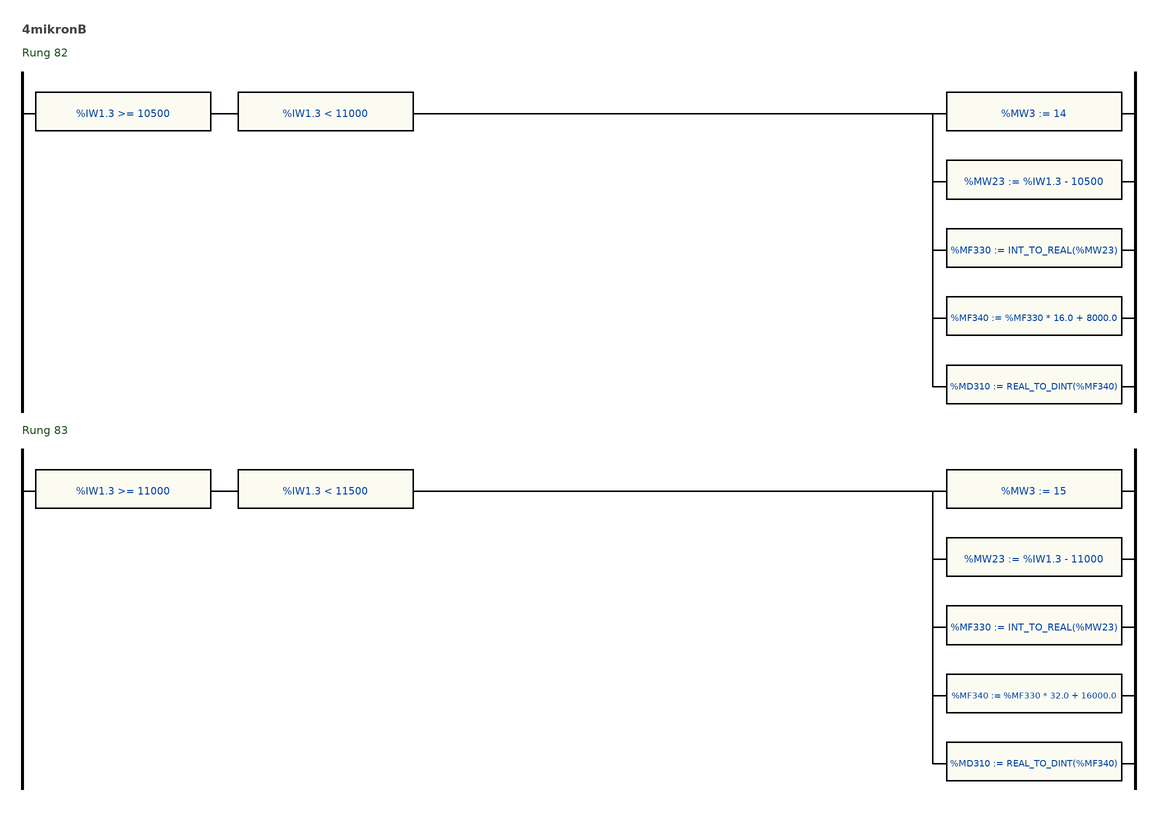

// Rung 82
  LD [ %IW1.3 >= 10500 ]
  AND [ %IW1.3 < 11000 ]
  [ %MW3 := 14 ]
  [ %MW23 := %IW1.3 - 10500 ]
  [ %MF330 := INT_TO_REAL ( %MW23 ) ]
  [ %MF340 := %MF330 * 16.0 + 8000.0 ]
  [ %MD310 := REAL_TO_DINT ( %MF340 ) ]
  // as ST:
  //   IF %IW1.3 >= 10500 AND %IW1.3 < 11000 THEN %MW3 := 14; END_IF;
  //   IF %IW1.3 >= 10500 AND %IW1.3 < 11000 THEN %MW23 := %IW1.3 - 10500; END_IF;
  //   IF %IW1.3 >= 10500 AND %IW1.3 < 11000 THEN %MF330 := INT_TO_REAL ( %MW23 ); END_IF;
  //   IF %IW1.3 >= 10500 AND %IW1.3 < 11000 THEN %MF340 := %MF330 * 16.0 + 8000.0; END_IF;
  //   IF %IW1.3 >= 10500 AND %IW1.3 < 11000 THEN %MD310 := REAL_TO_DINT ( %MF340 ); END_IF;

// Rung 83
  LD [ %IW1.3 >= 11000 ]
  AND [ %IW1.3 < 11500 ]
  [ %MW3 := 15 ]
  [ %MW23 := %IW1.3 - 11000 ]
  [ %MF330 := INT_TO_REAL ( %MW23 ) ]
  [ %MF340 := %MF330 * 32.0 + 16000.0 ]
  [ %MD310 := REAL_TO_DINT ( %MF340 ) ]
  // as ST:
  //   IF %IW1.3 >= 11000 AND %IW1.3 < 11500 THEN %MW3 := 15; END_IF;
  //   IF %IW1.3 >= 11000 AND %IW1.3 < 11500 THEN %MW23 := %IW1.3 - 11000; END_IF;
  //   IF %IW1.3 >= 11000 AND %IW1.3 < 11500 THEN %MF330 := INT_TO_REAL ( %MW23 ); END_IF;
  //   IF %IW1.3 >= 11000 AND %IW1.3 < 11500 THEN %MF340 := %MF330 * 32.0 + 16000.0; END_IF;
  //   IF %IW1.3 >= 11000 AND %IW1.3 < 11500 THEN %MD310 := REAL_TO_DINT ( %MF340 ); END_IF;

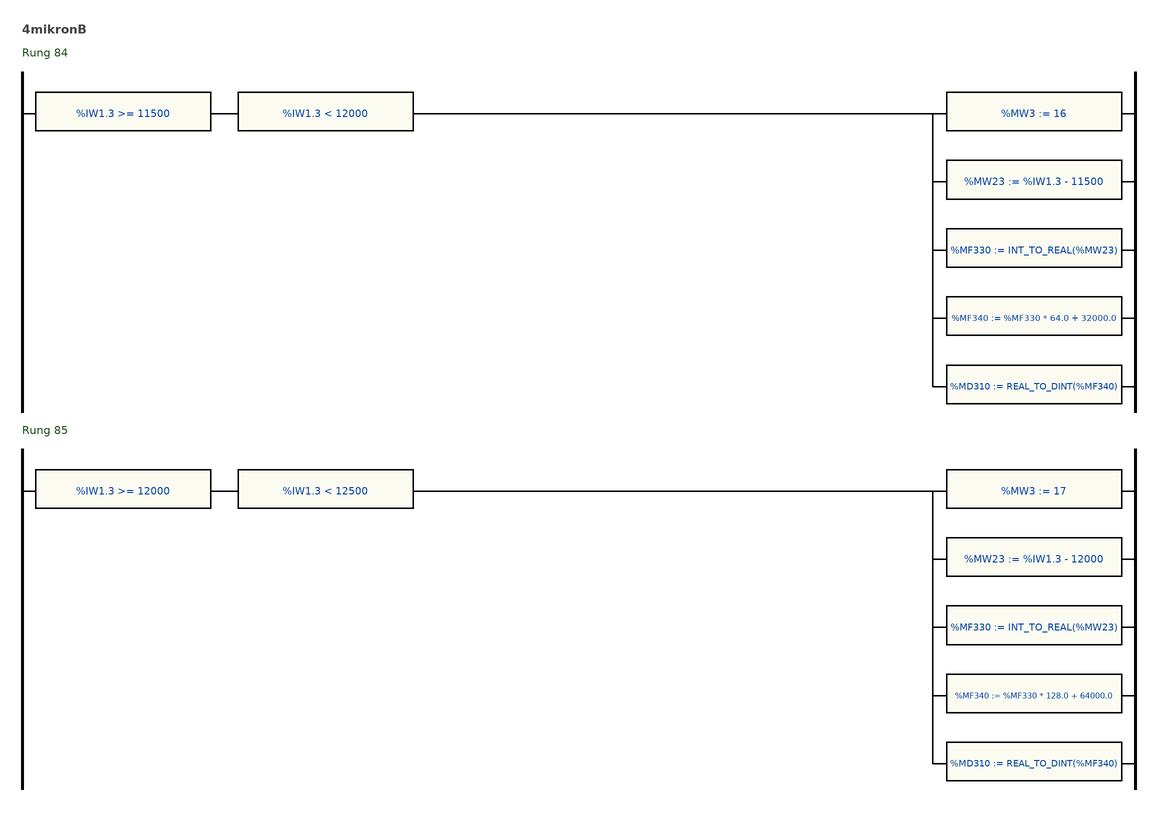

// Rung 84
  LD [ %IW1.3 >= 11500 ]
  AND [ %IW1.3 < 12000 ]
  [ %MW3 := 16 ]
  [ %MW23 := %IW1.3 - 11500 ]
  [ %MF330 := INT_TO_REAL ( %MW23 ) ]
  [ %MF340 := %MF330 * 64.0 + 32000.0 ]
  [ %MD310 := REAL_TO_DINT ( %MF340 ) ]
  // as ST:
  //   IF %IW1.3 >= 11500 AND %IW1.3 < 12000 THEN %MW3 := 16; END_IF;
  //   IF %IW1.3 >= 11500 AND %IW1.3 < 12000 THEN %MW23 := %IW1.3 - 11500; END_IF;
  //   IF %IW1.3 >= 11500 AND %IW1.3 < 12000 THEN %MF330 := INT_TO_REAL ( %MW23 ); END_IF;
  //   IF %IW1.3 >= 11500 AND %IW1.3 < 12000 THEN %MF340 := %MF330 * 64.0 + 32000.0; END_IF;
  //   IF %IW1.3 >= 11500 AND %IW1.3 < 12000 THEN %MD310 := REAL_TO_DINT ( %MF340 ); END_IF;

// Rung 85
  LD [ %IW1.3 >= 12000 ]
  AND [ %IW1.3 < 12500 ]
  [ %MW3 := 17 ]
  [ %MW23 := %IW1.3 - 12000 ]
  [ %MF330 := INT_TO_REAL ( %MW23 ) ]
  [ %MF340 := %MF330 * 128.0 + 64000.0 ]
  [ %MD310 := REAL_TO_DINT ( %MF340 ) ]
  // as ST:
  //   IF %IW1.3 >= 12000 AND %IW1.3 < 12500 THEN %MW3 := 17; END_IF;
  //   IF %IW1.3 >= 12000 AND %IW1.3 < 12500 THEN %MW23 := %IW1.3 - 12000; END_IF;
  //   IF %IW1.3 >= 12000 AND %IW1.3 < 12500 THEN %MF330 := INT_TO_REAL ( %MW23 ); END_IF;
  //   IF %IW1.3 >= 12000 AND %IW1.3 < 12500 THEN %MF340 := %MF330 * 128.0 + 64000.0; END_IF;
  //   IF %IW1.3 >= 12000 AND %IW1.3 < 12500 THEN %MD310 := REAL_TO_DINT ( %MF340 ); END_IF;

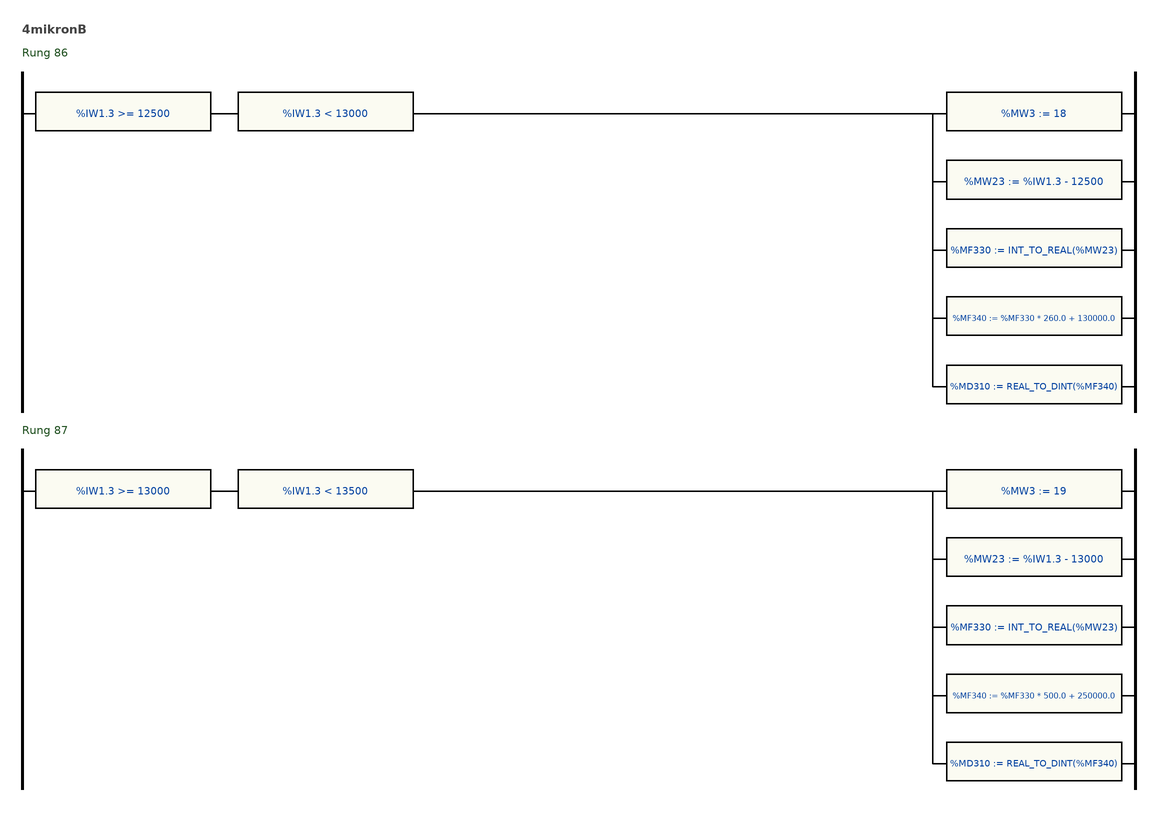

// Rung 86
  LD [ %IW1.3 >= 12500 ]
  AND [ %IW1.3 < 13000 ]
  [ %MW3 := 18 ]
  [ %MW23 := %IW1.3 - 12500 ]
  [ %MF330 := INT_TO_REAL ( %MW23 ) ]
  [ %MF340 := %MF330 * 260.0 + 130000.0 ]
  [ %MD310 := REAL_TO_DINT ( %MF340 ) ]
  // as ST:
  //   IF %IW1.3 >= 12500 AND %IW1.3 < 13000 THEN %MW3 := 18; END_IF;
  //   IF %IW1.3 >= 12500 AND %IW1.3 < 13000 THEN %MW23 := %IW1.3 - 12500; END_IF;
  //   IF %IW1.3 >= 12500 AND %IW1.3 < 13000 THEN %MF330 := INT_TO_REAL ( %MW23 ); END_IF;
  //   IF %IW1.3 >= 12500 AND %IW1.3 < 13000 THEN %MF340 := %MF330 * 260.0 + 130000.0; END_IF;
  //   IF %IW1.3 >= 12500 AND %IW1.3 < 13000 THEN %MD310 := REAL_TO_DINT ( %MF340 ); END_IF;

// Rung 87
  LD [ %IW1.3 >= 13000 ]
  AND [ %IW1.3 < 13500 ]
  [ %MW3 := 19 ]
  [ %MW23 := %IW1.3 - 13000 ]
  [ %MF330 := INT_TO_REAL ( %MW23 ) ]
  [ %MF340 := %MF330 * 500.0 + 250000.0 ]
  [ %MD310 := REAL_TO_DINT ( %MF340 ) ]
  // as ST:
  //   IF %IW1.3 >= 13000 AND %IW1.3 < 13500 THEN %MW3 := 19; END_IF;
  //   IF %IW1.3 >= 13000 AND %IW1.3 < 13500 THEN %MW23 := %IW1.3 - 13000; END_IF;
  //   IF %IW1.3 >= 13000 AND %IW1.3 < 13500 THEN %MF330 := INT_TO_REAL ( %MW23 ); END_IF;
  //   IF %IW1.3 >= 13000 AND %IW1.3 < 13500 THEN %MF340 := %MF330 * 500.0 + 250000.0; END_IF;
  //   IF %IW1.3 >= 13000 AND %IW1.3 < 13500 THEN %MD310 := REAL_TO_DINT ( %MF340 ); END_IF;

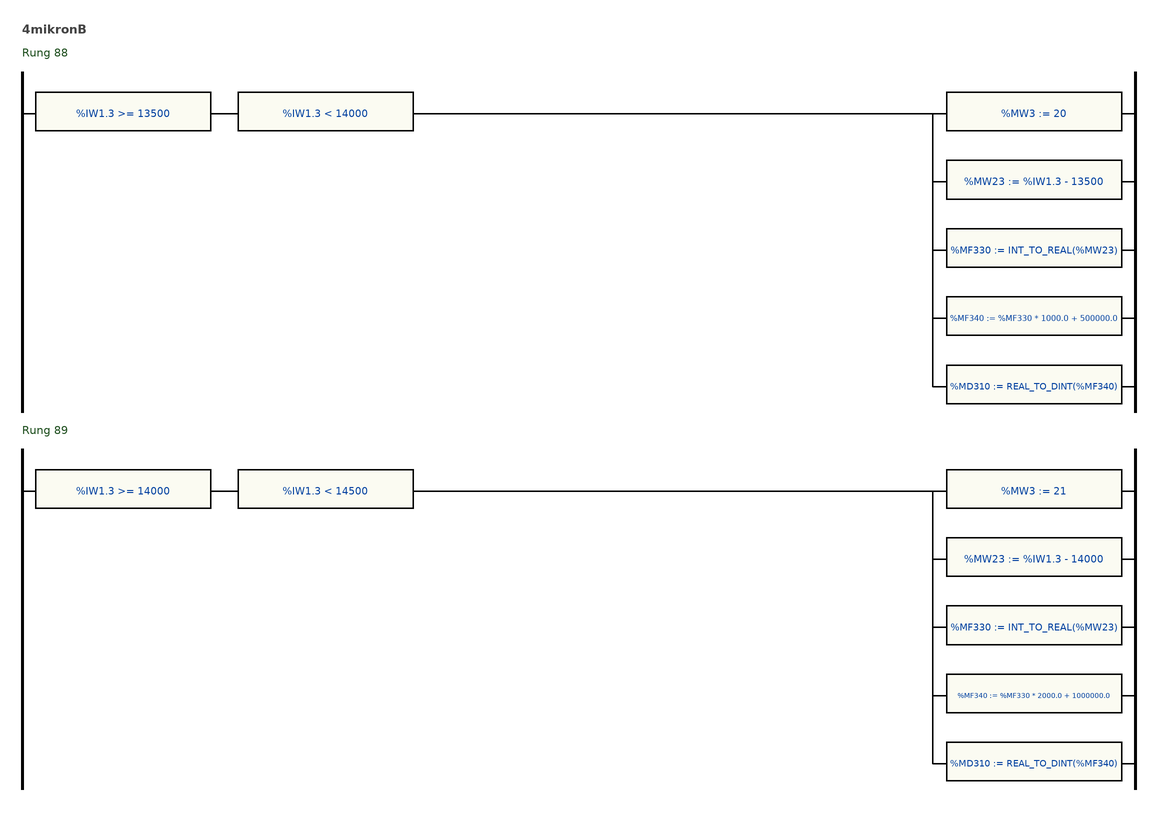

// Rung 88
  LD [ %IW1.3 >= 13500 ]
  AND [ %IW1.3 < 14000 ]
  [ %MW3 := 20 ]
  [ %MW23 := %IW1.3 - 13500 ]
  [ %MF330 := INT_TO_REAL ( %MW23 ) ]
  [ %MF340 := %MF330 * 1000.0 + 500000.0 ]
  [ %MD310 := REAL_TO_DINT ( %MF340 ) ]
  // as ST:
  //   IF %IW1.3 >= 13500 AND %IW1.3 < 14000 THEN %MW3 := 20; END_IF;
  //   IF %IW1.3 >= 13500 AND %IW1.3 < 14000 THEN %MW23 := %IW1.3 - 13500; END_IF;
  //   IF %IW1.3 >= 13500 AND %IW1.3 < 14000 THEN %MF330 := INT_TO_REAL ( %MW23 ); END_IF;
  //   IF %IW1.3 >= 13500 AND %IW1.3 < 14000 THEN %MF340 := %MF330 * 1000.0 + 500000.0; END_IF;
  //   IF %IW1.3 >= 13500 AND %IW1.3 < 14000 THEN %MD310 := REAL_TO_DINT ( %MF340 ); END_IF;

// Rung 89
  LD [ %IW1.3 >= 14000 ]
  AND [ %IW1.3 < 14500 ]
  [ %MW3 := 21 ]
  [ %MW23 := %IW1.3 - 14000 ]
  [ %MF330 := INT_TO_REAL ( %MW23 ) ]
  [ %MF340 := %MF330 * 2000.0 + 1000000.0 ]
  [ %MD310 := REAL_TO_DINT ( %MF340 ) ]
  // as ST:
  //   IF %IW1.3 >= 14000 AND %IW1.3 < 14500 THEN %MW3 := 21; END_IF;
  //   IF %IW1.3 >= 14000 AND %IW1.3 < 14500 THEN %MW23 := %IW1.3 - 14000; END_IF;
  //   IF %IW1.3 >= 14000 AND %IW1.3 < 14500 THEN %MF330 := INT_TO_REAL ( %MW23 ); END_IF;
  //   IF %IW1.3 >= 14000 AND %IW1.3 < 14500 THEN %MF340 := %MF330 * 2000.0 + 1000000.0; END_IF;
  //   IF %IW1.3 >= 14000 AND %IW1.3 < 14500 THEN %MD310 := REAL_TO_DINT ( %MF340 ); END_IF;

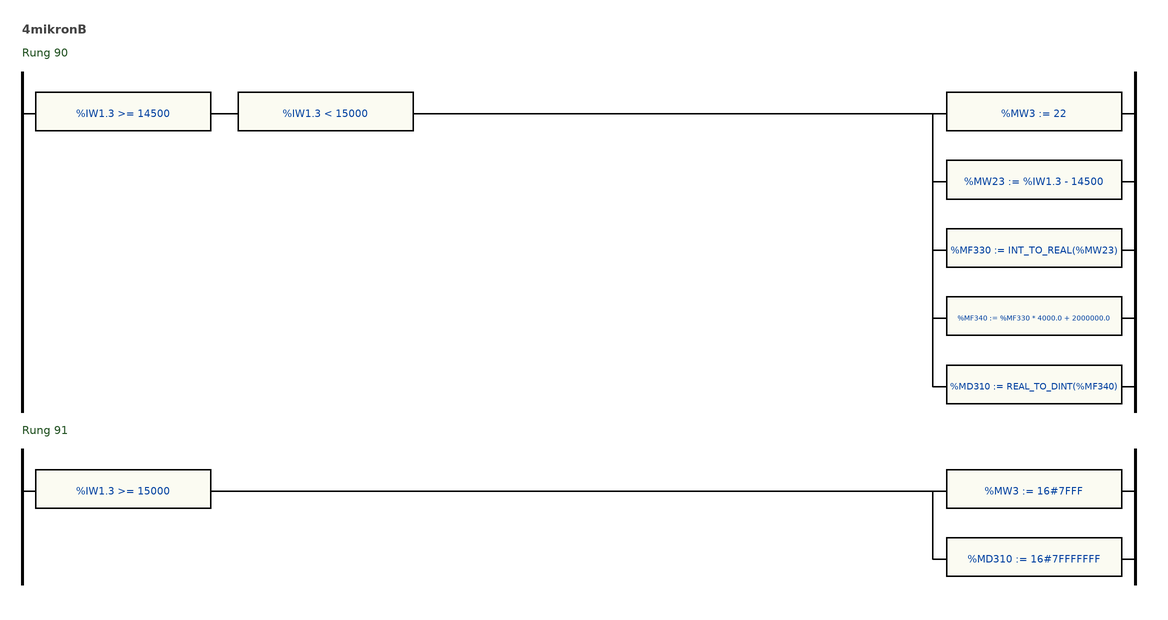

// Rung 90
  LD [ %IW1.3 >= 14500 ]
  AND [ %IW1.3 < 15000 ]
  [ %MW3 := 22 ]
  [ %MW23 := %IW1.3 - 14500 ]
  [ %MF330 := INT_TO_REAL ( %MW23 ) ]
  [ %MF340 := %MF330 * 4000.0 + 2000000.0 ]
  [ %MD310 := REAL_TO_DINT ( %MF340 ) ]
  // as ST:
  //   IF %IW1.3 >= 14500 AND %IW1.3 < 15000 THEN %MW3 := 22; END_IF;
  //   IF %IW1.3 >= 14500 AND %IW1.3 < 15000 THEN %MW23 := %IW1.3 - 14500; END_IF;
  //   IF %IW1.3 >= 14500 AND %IW1.3 < 15000 THEN %MF330 := INT_TO_REAL ( %MW23 ); END_IF;
  //   IF %IW1.3 >= 14500 AND %IW1.3 < 15000 THEN %MF340 := %MF330 * 4000.0 + 2000000.0; END_IF;
  //   IF %IW1.3 >= 14500 AND %IW1.3 < 15000 THEN %MD310 := REAL_TO_DINT ( %MF340 ); END_IF;

// Rung 91
  LD [ %IW1.3 >= 15000 ]
  [ %MW3 := 16#7FFF ]
  [ %MD310 := 16#7FFFFFFF ]
  // as ST:
  //   IF %IW1.3 >= 15000 THEN %MW3 := 16#7FFF; END_IF;
  //   IF %IW1.3 >= 15000 THEN %MD310 := 16#7FFFFFFF; END_IF;

POU 6mikronB
  (* SectionNumber=5 *)

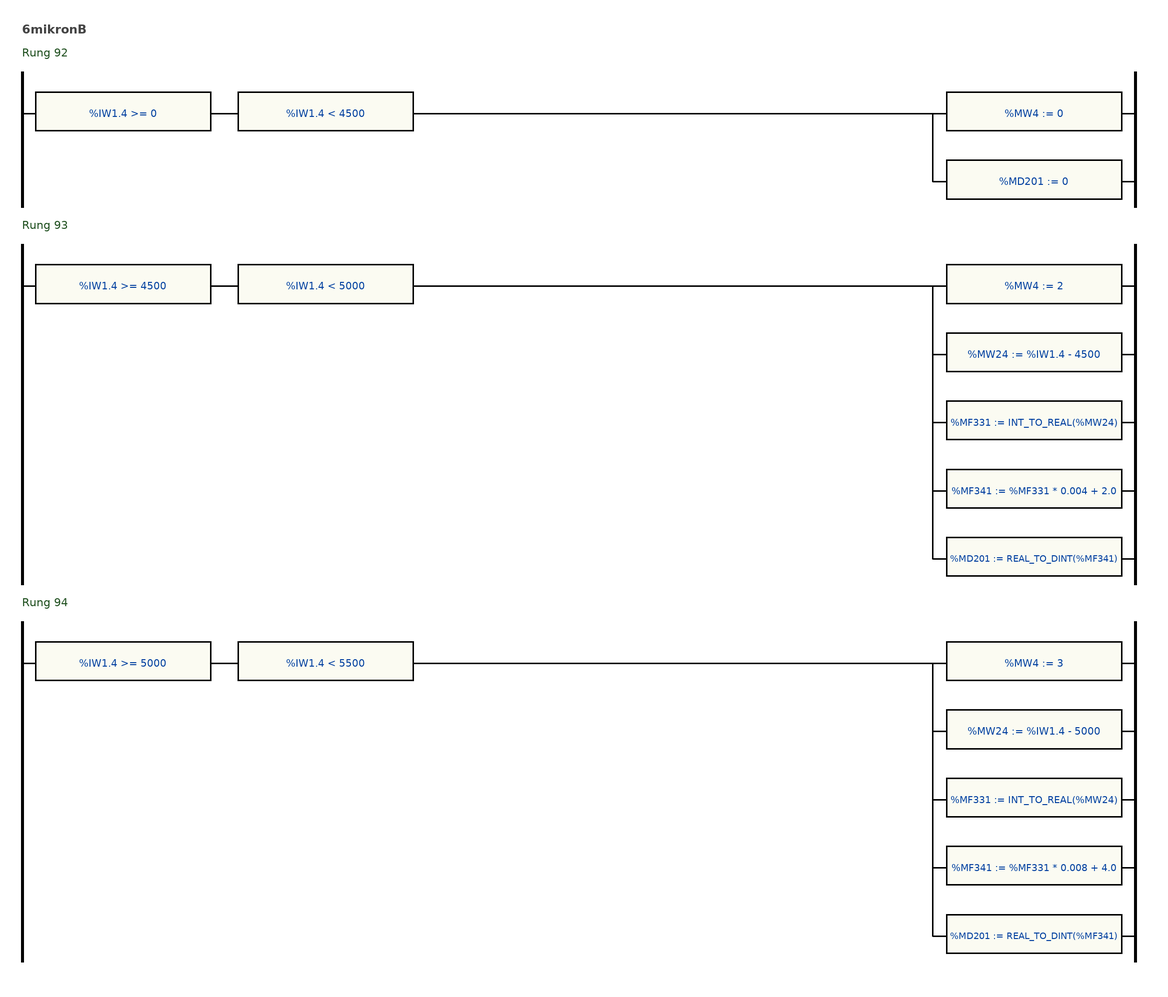

// Rung 92
  LD [ %IW1.4 >= 0 ]
  AND [ %IW1.4 < 4500 ]
  [ %MW4 := 0 ]
  [ %MD201 := 0 ]
  // as ST:
  //   IF %IW1.4 >= 0 AND %IW1.4 < 4500 THEN %MW4 := 0; END_IF;
  //   IF %IW1.4 >= 0 AND %IW1.4 < 4500 THEN %MD201 := 0; END_IF;

// Rung 93
  LD [ %IW1.4 >= 4500 ]
  AND [ %IW1.4 < 5000 ]
  [ %MW4 := 2 ]
  [ %MW24 := %IW1.4 - 4500 ]
  [ %MF331 := INT_TO_REAL ( %MW24 ) ]
  [ %MF341 := %MF331 * 0.004 + 2.0 ]
  [ %MD201 := REAL_TO_DINT ( %MF341 ) ]
  // as ST:
  //   IF %IW1.4 >= 4500 AND %IW1.4 < 5000 THEN %MW4 := 2; END_IF;
  //   IF %IW1.4 >= 4500 AND %IW1.4 < 5000 THEN %MW24 := %IW1.4 - 4500; END_IF;
  //   IF %IW1.4 >= 4500 AND %IW1.4 < 5000 THEN %MF331 := INT_TO_REAL ( %MW24 ); END_IF;
  //   IF %IW1.4 >= 4500 AND %IW1.4 < 5000 THEN %MF341 := %MF331 * 0.004 + 2.0; END_IF;
  //   IF %IW1.4 >= 4500 AND %IW1.4 < 5000 THEN %MD201 := REAL_TO_DINT ( %MF341 ); END_IF;

// Rung 94
  LD [ %IW1.4 >= 5000 ]
  AND [ %IW1.4 < 5500 ]
  [ %MW4 := 3 ]
  [ %MW24 := %IW1.4 - 5000 ]
  [ %MF331 := INT_TO_REAL ( %MW24 ) ]
  [ %MF341 := %MF331 * 0.008 + 4.0 ]
  [ %MD201 := REAL_TO_DINT ( %MF341 ) ]
  // as ST:
  //   IF %IW1.4 >= 5000 AND %IW1.4 < 5500 THEN %MW4 := 3; END_IF;
  //   IF %IW1.4 >= 5000 AND %IW1.4 < 5500 THEN %MW24 := %IW1.4 - 5000; END_IF;
  //   IF %IW1.4 >= 5000 AND %IW1.4 < 5500 THEN %MF331 := INT_TO_REAL ( %MW24 ); END_IF;
  //   IF %IW1.4 >= 5000 AND %IW1.4 < 5500 THEN %MF341 := %MF331 * 0.008 + 4.0; END_IF;
  //   IF %IW1.4 >= 5000 AND %IW1.4 < 5500 THEN %MD201 := REAL_TO_DINT ( %MF341 ); END_IF;

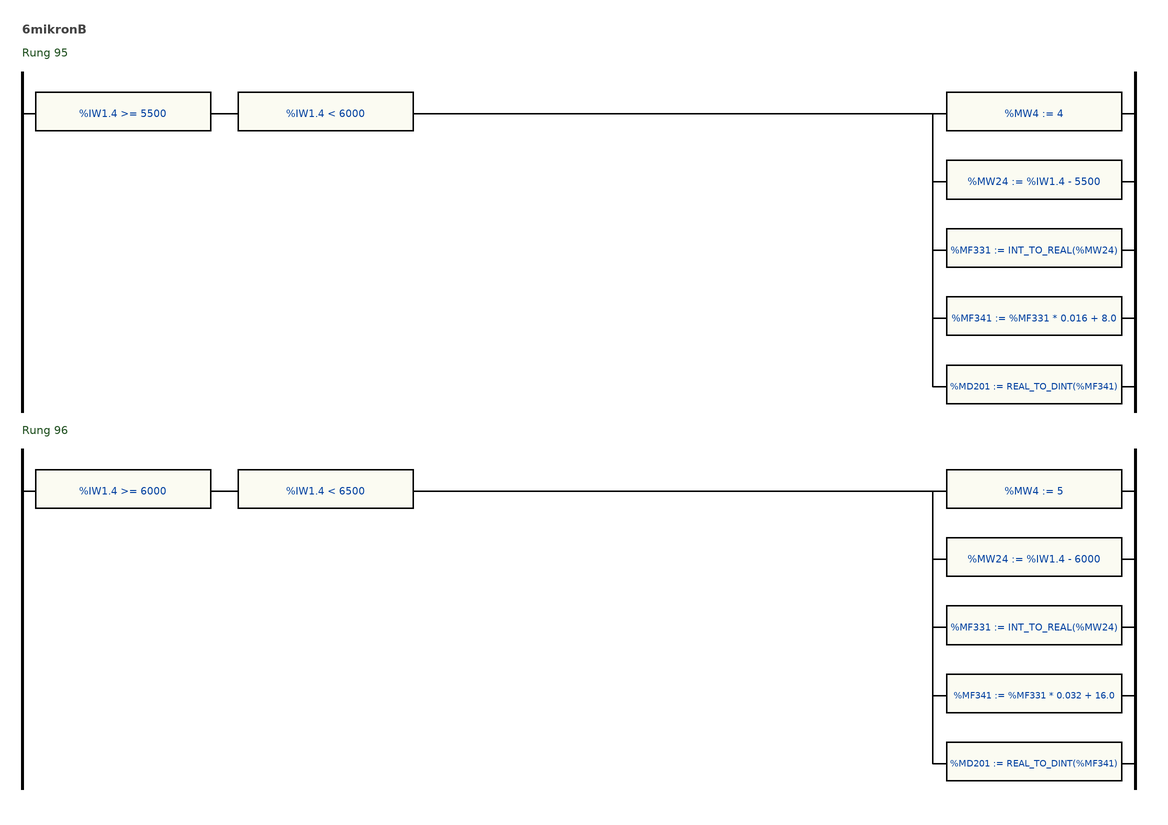

// Rung 95
  LD [ %IW1.4 >= 5500 ]
  AND [ %IW1.4 < 6000 ]
  [ %MW4 := 4 ]
  [ %MW24 := %IW1.4 - 5500 ]
  [ %MF331 := INT_TO_REAL ( %MW24 ) ]
  [ %MF341 := %MF331 * 0.016 + 8.0 ]
  [ %MD201 := REAL_TO_DINT ( %MF341 ) ]
  // as ST:
  //   IF %IW1.4 >= 5500 AND %IW1.4 < 6000 THEN %MW4 := 4; END_IF;
  //   IF %IW1.4 >= 5500 AND %IW1.4 < 6000 THEN %MW24 := %IW1.4 - 5500; END_IF;
  //   IF %IW1.4 >= 5500 AND %IW1.4 < 6000 THEN %MF331 := INT_TO_REAL ( %MW24 ); END_IF;
  //   IF %IW1.4 >= 5500 AND %IW1.4 < 6000 THEN %MF341 := %MF331 * 0.016 + 8.0; END_IF;
  //   IF %IW1.4 >= 5500 AND %IW1.4 < 6000 THEN %MD201 := REAL_TO_DINT ( %MF341 ); END_IF;

// Rung 96
  LD [ %IW1.4 >= 6000 ]
  AND [ %IW1.4 < 6500 ]
  [ %MW4 := 5 ]
  [ %MW24 := %IW1.4 - 6000 ]
  [ %MF331 := INT_TO_REAL ( %MW24 ) ]
  [ %MF341 := %MF331 * 0.032 + 16.0 ]
  [ %MD201 := REAL_TO_DINT ( %MF341 ) ]
  // as ST:
  //   IF %IW1.4 >= 6000 AND %IW1.4 < 6500 THEN %MW4 := 5; END_IF;
  //   IF %IW1.4 >= 6000 AND %IW1.4 < 6500 THEN %MW24 := %IW1.4 - 6000; END_IF;
  //   IF %IW1.4 >= 6000 AND %IW1.4 < 6500 THEN %MF331 := INT_TO_REAL ( %MW24 ); END_IF;
  //   IF %IW1.4 >= 6000 AND %IW1.4 < 6500 THEN %MF341 := %MF331 * 0.032 + 16.0; END_IF;
  //   IF %IW1.4 >= 6000 AND %IW1.4 < 6500 THEN %MD201 := REAL_TO_DINT ( %MF341 ); END_IF;

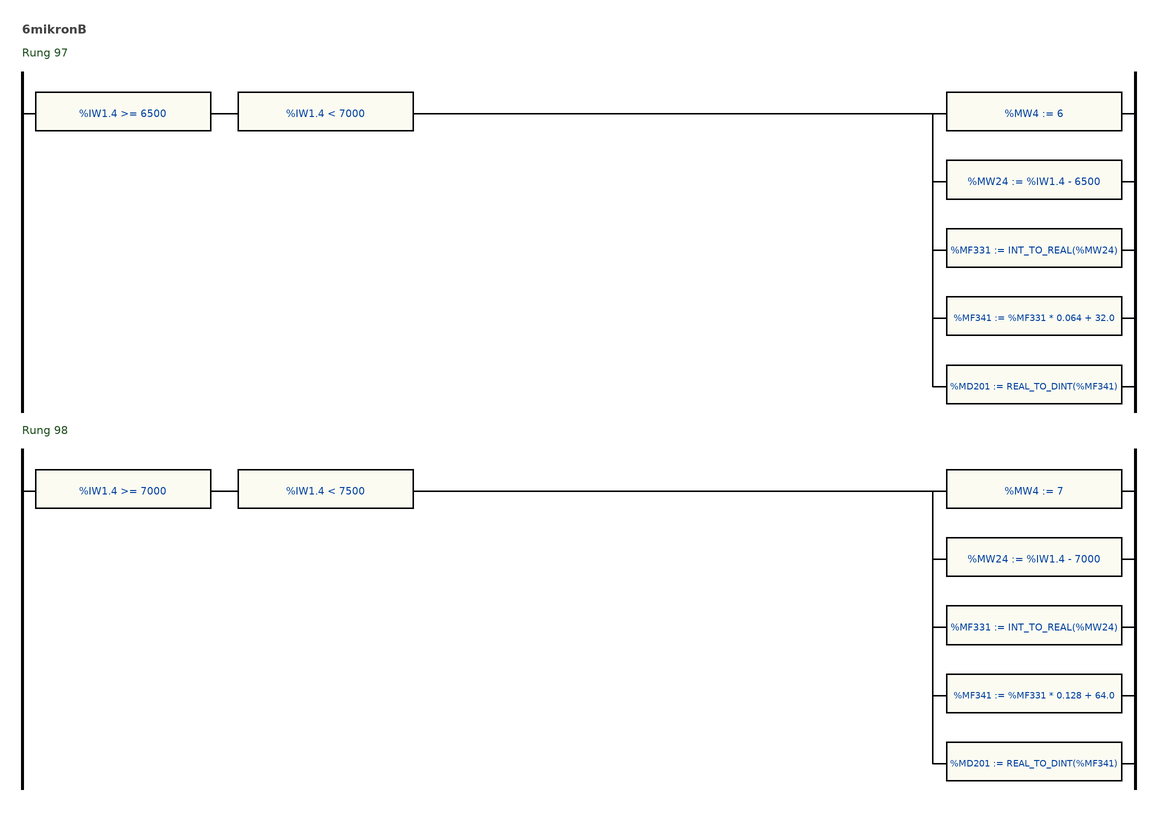

// Rung 97
  LD [ %IW1.4 >= 6500 ]
  AND [ %IW1.4 < 7000 ]
  [ %MW4 := 6 ]
  [ %MW24 := %IW1.4 - 6500 ]
  [ %MF331 := INT_TO_REAL ( %MW24 ) ]
  [ %MF341 := %MF331 * 0.064 + 32.0 ]
  [ %MD201 := REAL_TO_DINT ( %MF341 ) ]
  // as ST:
  //   IF %IW1.4 >= 6500 AND %IW1.4 < 7000 THEN %MW4 := 6; END_IF;
  //   IF %IW1.4 >= 6500 AND %IW1.4 < 7000 THEN %MW24 := %IW1.4 - 6500; END_IF;
  //   IF %IW1.4 >= 6500 AND %IW1.4 < 7000 THEN %MF331 := INT_TO_REAL ( %MW24 ); END_IF;
  //   IF %IW1.4 >= 6500 AND %IW1.4 < 7000 THEN %MF341 := %MF331 * 0.064 + 32.0; END_IF;
  //   IF %IW1.4 >= 6500 AND %IW1.4 < 7000 THEN %MD201 := REAL_TO_DINT ( %MF341 ); END_IF;

// Rung 98
  LD [ %IW1.4 >= 7000 ]
  AND [ %IW1.4 < 7500 ]
  [ %MW4 := 7 ]
  [ %MW24 := %IW1.4 - 7000 ]
  [ %MF331 := INT_TO_REAL ( %MW24 ) ]
  [ %MF341 := %MF331 * 0.128 + 64.0 ]
  [ %MD201 := REAL_TO_DINT ( %MF341 ) ]
  // as ST:
  //   IF %IW1.4 >= 7000 AND %IW1.4 < 7500 THEN %MW4 := 7; END_IF;
  //   IF %IW1.4 >= 7000 AND %IW1.4 < 7500 THEN %MW24 := %IW1.4 - 7000; END_IF;
  //   IF %IW1.4 >= 7000 AND %IW1.4 < 7500 THEN %MF331 := INT_TO_REAL ( %MW24 ); END_IF;
  //   IF %IW1.4 >= 7000 AND %IW1.4 < 7500 THEN %MF341 := %MF331 * 0.128 + 64.0; END_IF;
  //   IF %IW1.4 >= 7000 AND %IW1.4 < 7500 THEN %MD201 := REAL_TO_DINT ( %MF341 ); END_IF;

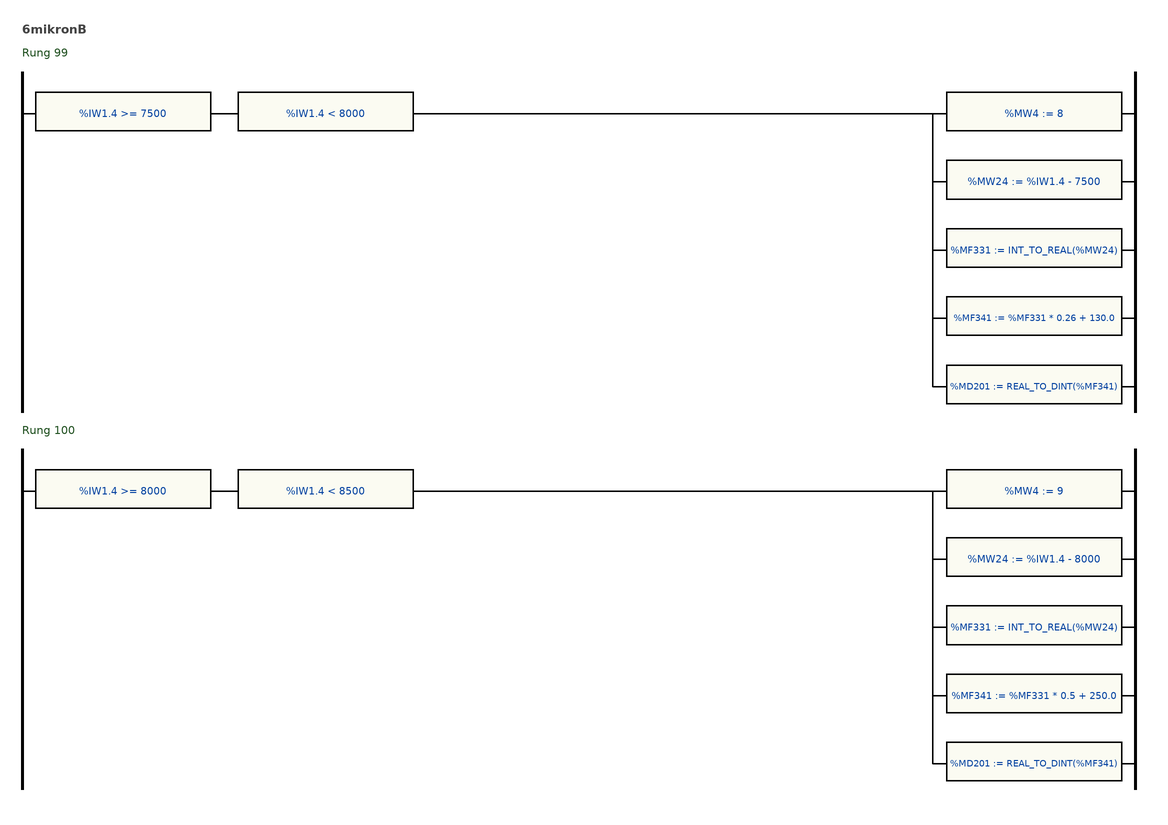

// Rung 99
  LD [ %IW1.4 >= 7500 ]
  AND [ %IW1.4 < 8000 ]
  [ %MW4 := 8 ]
  [ %MW24 := %IW1.4 - 7500 ]
  [ %MF331 := INT_TO_REAL ( %MW24 ) ]
  [ %MF341 := %MF331 * 0.26 + 130.0 ]
  [ %MD201 := REAL_TO_DINT ( %MF341 ) ]
  // as ST:
  //   IF %IW1.4 >= 7500 AND %IW1.4 < 8000 THEN %MW4 := 8; END_IF;
  //   IF %IW1.4 >= 7500 AND %IW1.4 < 8000 THEN %MW24 := %IW1.4 - 7500; END_IF;
  //   IF %IW1.4 >= 7500 AND %IW1.4 < 8000 THEN %MF331 := INT_TO_REAL ( %MW24 ); END_IF;
  //   IF %IW1.4 >= 7500 AND %IW1.4 < 8000 THEN %MF341 := %MF331 * 0.26 + 130.0; END_IF;
  //   IF %IW1.4 >= 7500 AND %IW1.4 < 8000 THEN %MD201 := REAL_TO_DINT ( %MF341 ); END_IF;

// Rung 100
  LD [ %IW1.4 >= 8000 ]
  AND [ %IW1.4 < 8500 ]
  [ %MW4 := 9 ]
  [ %MW24 := %IW1.4 - 8000 ]
  [ %MF331 := INT_TO_REAL ( %MW24 ) ]
  [ %MF341 := %MF331 * 0.5 + 250.0 ]
  [ %MD201 := REAL_TO_DINT ( %MF341 ) ]
  // as ST:
  //   IF %IW1.4 >= 8000 AND %IW1.4 < 8500 THEN %MW4 := 9; END_IF;
  //   IF %IW1.4 >= 8000 AND %IW1.4 < 8500 THEN %MW24 := %IW1.4 - 8000; END_IF;
  //   IF %IW1.4 >= 8000 AND %IW1.4 < 8500 THEN %MF331 := INT_TO_REAL ( %MW24 ); END_IF;
  //   IF %IW1.4 >= 8000 AND %IW1.4 < 8500 THEN %MF341 := %MF331 * 0.5 + 250.0; END_IF;
  //   IF %IW1.4 >= 8000 AND %IW1.4 < 8500 THEN %MD201 := REAL_TO_DINT ( %MF341 ); END_IF;

